   1:  PR[GP1:91,1] = PR[GP1:90,1] + -0.145;
   1:  PR[GP1:91,2] = PR[GP1:90,2] + -15.711;
   1:L PR[91] 10mm/sec CNT100;
   1:  PR[GP1:91,1] = PR[GP1:90,1] + 0.024;
   1:  PR[GP1:91,2] = PR[GP1:90,2] + -15.638;
   1:L PR[91] 10mm/sec CNT100;
   1:  PR[GP1:91,1] = PR[GP1:90,1] + 0.412;
   1:  PR[GP1:91,2] = PR[GP1:90,2] + -15.609;
   1:L PR[91] 10mm/sec CNT100;
   1:  PR[GP1:91,1] = PR[GP1:90,1] + 1.712;
   1:  PR[GP1:91,2] = PR[GP1:90,2] + -16.090;
   1:L PR[91] 10mm/sec CNT100;
   1:  PR[GP1:91,1] = PR[GP1:90,1] + 2.427;
   1:  PR[GP1:91,2] = PR[GP1:90,2] + -16.554;
   1:L PR[91] 10mm/sec CNT100;
   1:  PR[GP1:91,1] = PR[GP1:90,1] + 3.285;
   1:  PR[GP1:91,2] = PR[GP1:90,2] + -17.042;
   1:L PR[91] 10mm/sec CNT100;
   1:  PR[GP1:91,1] = PR[GP1:90,1] + 4.793;
   1:  PR[GP1:91,2] = PR[GP1:90,2] + -17.836;
   1:L PR[91] 10mm/sec CNT100;
   1:  PR[GP1:91,1] = PR[GP1:90,1] + 5.956;
   1:  PR[GP1:91,2] = PR[GP1:90,2] + -18.277;
   1:L PR[91] 10mm/sec CNT100;
   1:  PR[GP1:91,1] = PR[GP1:90,1] + 7.268;
   1:  PR[GP1:91,2] = PR[GP1:90,2] + -18.717;
   1:L PR[91] 10mm/sec CNT100;
   1:  PR[GP1:91,1] = PR[GP1:90,1] + 8.896;
   1:  PR[GP1:91,2] = PR[GP1:90,2] + -19.063;
   1:L PR[91] 10mm/sec CNT100;
   1:  PR[GP1:91,1] = PR[GP1:90,1] + 9.804;
   1:  PR[GP1:91,2] = PR[GP1:90,2] + -19.215;
   1:L PR[91] 10mm/sec CNT100;
   1:  PR[GP1:91,1] = PR[GP1:90,1] + 12.012;
   1:  PR[GP1:91,2] = PR[GP1:90,2] + -19.347;
   1:L PR[91] 10mm/sec CNT100;
   1:  PR[GP1:91,1] = PR[GP1:90,1] + 12.321;
   1:  PR[GP1:91,2] = PR[GP1:90,2] + -19.350;
   1:L PR[91] 10mm/sec CNT100;
   1:  PR[GP1:91,1] = PR[GP1:90,1] + 13.545;
   1:  PR[GP1:91,2] = PR[GP1:90,2] + -19.242;
   1:L PR[91] 10mm/sec CNT100;
   1:  PR[GP1:91,1] = PR[GP1:90,1] + 14.916;
   1:  PR[GP1:91,2] = PR[GP1:90,2] + -19.147;
   1:L PR[91] 10mm/sec CNT100;
   1:  PR[GP1:91,1] = PR[GP1:90,1] + 17.562;
   1:  PR[GP1:91,2] = PR[GP1:90,2] + -18.593;
   1:L PR[91] 10mm/sec CNT100;
   1:  PR[GP1:91,1] = PR[GP1:90,1] + 19.003;
   1:  PR[GP1:91,2] = PR[GP1:90,2] + -18.092;
   1:L PR[91] 10mm/sec CNT100;
   1:  PR[GP1:91,1] = PR[GP1:90,1] + 20.123;
   1:  PR[GP1:91,2] = PR[GP1:90,2] + -17.685;
   1:L PR[91] 10mm/sec CNT100;
   1:  PR[GP1:91,1] = PR[GP1:90,1] + 22.568;
   1:  PR[GP1:91,2] = PR[GP1:90,2] + -16.427;
   1:L PR[91] 10mm/sec CNT100;
   1:  PR[GP1:91,1] = PR[GP1:90,1] + 24.867;
   1:  PR[GP1:91,2] = PR[GP1:90,2] + -14.882;
   1:L PR[91] 10mm/sec CNT100;
   1:  PR[GP1:91,1] = PR[GP1:90,1] + 25.707;
   1:  PR[GP1:91,2] = PR[GP1:90,2] + -14.143;
   1:L PR[91] 10mm/sec CNT100;
   1:  PR[GP1:91,1] = PR[GP1:90,1] + 26.925;
   1:  PR[GP1:91,2] = PR[GP1:90,2] + -13.045;
   1:L PR[91] 10mm/sec CNT100;
   1:  PR[GP1:91,1] = PR[GP1:90,1] + 28.700;
   1:  PR[GP1:91,2] = PR[GP1:90,2] + -10.934;
   1:L PR[91] 10mm/sec CNT100;
   1:  PR[GP1:91,1] = PR[GP1:90,1] + 30.141;
   1:  PR[GP1:91,2] = PR[GP1:90,2] + -8.600;
   1:L PR[91] 10mm/sec CNT100;
   1:  PR[GP1:91,1] = PR[GP1:90,1] + 31.207;
   1:  PR[GP1:91,2] = PR[GP1:90,2] + -6.109;
   1:L PR[91] 10mm/sec CNT100;
   1:  PR[GP1:91,1] = PR[GP1:90,1] + 31.857;
   1:  PR[GP1:91,2] = PR[GP1:90,2] + -3.509;
   1:L PR[91] 10mm/sec CNT100;
   1:  PR[GP1:91,1] = PR[GP1:90,1] + 32.061;
   1:  PR[GP1:91,2] = PR[GP1:90,2] + -0.854;
   1:L PR[91] 10mm/sec CNT100;
   1:  PR[GP1:91,1] = PR[GP1:90,1] + 31.675;
   1:  PR[GP1:91,2] = PR[GP1:90,2] + 2.503;
   1:L PR[91] 10mm/sec CNT100;
   1:  PR[GP1:91,1] = PR[GP1:90,1] + 30.594;
   1:  PR[GP1:91,2] = PR[GP1:90,2] + 5.692;
   1:L PR[91] 10mm/sec CNT100;
   1:  PR[GP1:91,1] = PR[GP1:90,1] + 28.845;
   1:  PR[GP1:91,2] = PR[GP1:90,2] + 8.602;
   1:L PR[91] 10mm/sec CNT100;
   1:  PR[GP1:91,1] = PR[GP1:90,1] + 26.495;
   1:  PR[GP1:91,2] = PR[GP1:90,2] + 11.109;
   1:L PR[91] 10mm/sec CNT100;
   1:  PR[GP1:91,1] = PR[GP1:90,1] + 23.637;
   1:  PR[GP1:91,2] = PR[GP1:90,2] + 13.130;
   1:L PR[91] 10mm/sec CNT100;
   1:  PR[GP1:91,1] = PR[GP1:90,1] + 20.377;
   1:  PR[GP1:91,2] = PR[GP1:90,2] + 14.590;
   1:L PR[91] 10mm/sec CNT100;
   1:  PR[GP1:91,1] = PR[GP1:90,1] + 16.885;
   1:  PR[GP1:91,2] = PR[GP1:90,2] + 15.406;
   1:L PR[91] 10mm/sec CNT100;
   1:  PR[GP1:91,1] = PR[GP1:90,1] + 14.816;
   1:  PR[GP1:91,2] = PR[GP1:90,2] + 15.503;
   1:L PR[91] 10mm/sec CNT100;
   1:  PR[GP1:91,1] = PR[GP1:90,1] + 13.268;
   1:  PR[GP1:91,2] = PR[GP1:90,2] + 15.568;
   1:L PR[91] 10mm/sec CNT100;
   1:  PR[GP1:91,1] = PR[GP1:90,1] + 9.649;
   1:  PR[GP1:91,2] = PR[GP1:90,2] + 15.081;
   1:L PR[91] 10mm/sec CNT100;
   1:  PR[GP1:91,1] = PR[GP1:90,1] + 6.237;
   1:  PR[GP1:91,2] = PR[GP1:90,2] + 13.936;
   1:L PR[91] 10mm/sec CNT100;
   1:  PR[GP1:91,1] = PR[GP1:90,1] + 3.041;
   1:  PR[GP1:91,2] = PR[GP1:90,2] + 12.211;
   1:L PR[91] 10mm/sec CNT100;
   1:  PR[GP1:91,1] = PR[GP1:90,1] + 1.090;
   1:  PR[GP1:91,2] = PR[GP1:90,2] + 10.690;
   1:L PR[91] 10mm/sec CNT100;
   1:  PR[GP1:91,1] = PR[GP1:90,1] + -0.001;
   1:  PR[GP1:91,2] = PR[GP1:90,2] + 10.133;
   1:L PR[91] 10mm/sec CNT100;
   1:  PR[GP1:91,1] = PR[GP1:90,1] + -1.282;
   1:  PR[GP1:91,2] = PR[GP1:90,2] + 10.163;
   1:L PR[91] 10mm/sec CNT100;
   1:  PR[GP1:91,1] = PR[GP1:90,1] + -2.059;
   1:  PR[GP1:91,2] = PR[GP1:90,2] + 10.540;
   1:L PR[91] 10mm/sec CNT100;
   1:  PR[GP1:91,1] = PR[GP1:90,1] + -3.147;
   1:  PR[GP1:91,2] = PR[GP1:90,2] + 11.202;
   1:L PR[91] 10mm/sec CNT100;
   1:  PR[GP1:91,1] = PR[GP1:90,1] + -4.530;
   1:  PR[GP1:91,2] = PR[GP1:90,2] + 12.155;
   1:L PR[91] 10mm/sec CNT100;
   1:  PR[GP1:91,1] = PR[GP1:90,1] + -5.421;
   1:  PR[GP1:91,2] = PR[GP1:90,2] + 12.681;
   1:L PR[91] 10mm/sec CNT100;
   1:  PR[GP1:91,1] = PR[GP1:90,1] + -7.191;
   1:  PR[GP1:91,2] = PR[GP1:90,2] + 13.488;
   1:L PR[91] 10mm/sec CNT100;
   1:  PR[GP1:91,1] = PR[GP1:90,1] + -9.797;
   1:  PR[GP1:91,2] = PR[GP1:90,2] + 14.446;
   1:L PR[91] 10mm/sec CNT100;
   1:  PR[GP1:91,1] = PR[GP1:90,1] + -10.237;
   1:  PR[GP1:91,2] = PR[GP1:90,2] + 14.563;
   1:L PR[91] 10mm/sec CNT100;
   1:  PR[GP1:91,1] = PR[GP1:90,1] + -13.368;
   1:  PR[GP1:91,2] = PR[GP1:90,2] + 15.140;
   1:L PR[91] 10mm/sec CNT100;
   1:  PR[GP1:91,1] = PR[GP1:90,1] + -14.004;
   1:  PR[GP1:91,2] = PR[GP1:90,2] + 15.238;
   1:L PR[91] 10mm/sec CNT100;
   1:  PR[GP1:91,1] = PR[GP1:90,1] + -16.372;
   1:  PR[GP1:91,2] = PR[GP1:90,2] + 15.227;
   1:L PR[91] 10mm/sec CNT100;
   1:  PR[GP1:91,1] = PR[GP1:90,1] + -17.931;
   1:  PR[GP1:91,2] = PR[GP1:90,2] + 15.176;
   1:L PR[91] 10mm/sec CNT100;
   1:  PR[GP1:91,1] = PR[GP1:90,1] + -19.411;
   1:  PR[GP1:91,2] = PR[GP1:90,2] + 14.876;
   1:L PR[91] 10mm/sec CNT100;
   1:  PR[GP1:91,1] = PR[GP1:90,1] + -21.644;
   1:  PR[GP1:91,2] = PR[GP1:90,2] + 14.370;
   1:L PR[91] 10mm/sec CNT100;
   1:  PR[GP1:91,1] = PR[GP1:90,1] + -22.403;
   1:  PR[GP1:91,2] = PR[GP1:90,2] + 14.049;
   1:L PR[91] 10mm/sec CNT100;
   1:  PR[GP1:91,1] = PR[GP1:90,1] + -25.006;
   1:  PR[GP1:91,2] = PR[GP1:90,2] + 12.891;
   1:L PR[91] 10mm/sec CNT100;
   1:  PR[GP1:91,1] = PR[GP1:90,1] + -27.897;
   1:  PR[GP1:91,2] = PR[GP1:90,2] + 10.819;
   1:L PR[91] 10mm/sec CNT100;
   1:  PR[GP1:91,1] = PR[GP1:90,1] + -30.164;
   1:  PR[GP1:91,2] = PR[GP1:90,2] + 8.232;
   1:L PR[91] 10mm/sec CNT100;
   1:  PR[GP1:91,1] = PR[GP1:90,1] + -31.840;
   1:  PR[GP1:91,2] = PR[GP1:90,2] + 5.244;
   1:L PR[91] 10mm/sec CNT100;
   1:  PR[GP1:91,1] = PR[GP1:90,1] + -32.875;
   1:  PR[GP1:91,2] = PR[GP1:90,2] + 1.996;
   1:L PR[91] 10mm/sec CNT100;
   1:  PR[GP1:91,1] = PR[GP1:90,1] + -33.174;
   1:  PR[GP1:91,2] = PR[GP1:90,2] + -1.394;
   1:L PR[91] 10mm/sec CNT100;
   1:  PR[GP1:91,1] = PR[GP1:90,1] + -33.130;
   1:  PR[GP1:91,2] = PR[GP1:90,2] + -1.625;
   1:L PR[91] 10mm/sec CNT100;
   1:  PR[GP1:91,1] = PR[GP1:90,1] + -32.704;
   1:  PR[GP1:91,2] = PR[GP1:90,2] + -4.886;
   1:L PR[91] 10mm/sec CNT100;
   1:  PR[GP1:91,1] = PR[GP1:90,1] + -32.550;
   1:  PR[GP1:91,2] = PR[GP1:90,2] + -5.342;
   1:L PR[91] 10mm/sec CNT100;
   1:  PR[GP1:91,1] = PR[GP1:90,1] + -31.594;
   1:  PR[GP1:91,2] = PR[GP1:90,2] + -7.989;
   1:L PR[91] 10mm/sec CNT100;
   1:  PR[GP1:91,1] = PR[GP1:90,1] + -31.506;
   1:  PR[GP1:91,2] = PR[GP1:90,2] + -8.224;
   1:L PR[91] 10mm/sec CNT100;
   1:  PR[GP1:91,1] = PR[GP1:90,1] + -29.951;
   1:  PR[GP1:91,2] = PR[GP1:90,2] + -10.706;
   1:L PR[91] 10mm/sec CNT100;
   1:  PR[GP1:91,1] = PR[GP1:90,1] + -29.521;
   1:  PR[GP1:91,2] = PR[GP1:90,2] + -11.361;
   1:L PR[91] 10mm/sec CNT100;
   1:  PR[GP1:91,1] = PR[GP1:90,1] + -27.878;
   1:  PR[GP1:91,2] = PR[GP1:90,2] + -13.093;
   1:L PR[91] 10mm/sec CNT100;
   1:  PR[GP1:91,1] = PR[GP1:90,1] + -26.835;
   1:  PR[GP1:91,2] = PR[GP1:90,2] + -14.134;
   1:L PR[91] 10mm/sec CNT100;
   1:  PR[GP1:91,1] = PR[GP1:90,1] + -25.477;
   1:  PR[GP1:91,2] = PR[GP1:90,2] + -15.103;
   1:L PR[91] 10mm/sec CNT100;
   1:  PR[GP1:91,1] = PR[GP1:90,1] + -22.956;
   1:  PR[GP1:91,2] = PR[GP1:90,2] + -16.602;
   1:  PR[GP1:91,3] = PR[GP1:90,3] + 26.400;
   1:L PR[91] 10mm/sec CNT100;
   1:  PR[GP1:91,1] = PR[GP1:90,1] + -19.409;
   1:  PR[GP1:91,2] = PR[GP1:90,2] + -18.084;
   1:L PR[91] 10mm/sec CNT100;
   1:  PR[GP1:91,1] = PR[GP1:90,1] + -17.838;
   1:  PR[GP1:91,2] = PR[GP1:90,2] + -18.496;
   1:L PR[91] 10mm/sec CNT100;
   1:  PR[GP1:91,1] = PR[GP1:90,1] + -15.882;
   1:  PR[GP1:91,2] = PR[GP1:90,2] + -18.925;
   1:L PR[91] 10mm/sec CNT100;
   1:  PR[GP1:91,1] = PR[GP1:90,1] + -12.351;
   1:  PR[GP1:91,2] = PR[GP1:90,2] + -19.223;
   1:L PR[91] 10mm/sec CNT100;
   1:  PR[GP1:91,1] = PR[GP1:90,1] + -9.475;
   1:  PR[GP1:91,2] = PR[GP1:90,2] + -19.059;
   1:L PR[91] 10mm/sec CNT100;
   1:  PR[GP1:91,1] = PR[GP1:90,1] + -8.254;
   1:  PR[GP1:91,2] = PR[GP1:90,2] + -18.972;
   1:L PR[91] 10mm/sec CNT100;
   1:  PR[GP1:91,1] = PR[GP1:90,1] + -5.076;
   1:  PR[GP1:91,2] = PR[GP1:90,2] + -18.282;
   1:L PR[91] 10mm/sec CNT100;
   1:  PR[GP1:91,1] = PR[GP1:90,1] + -2.226;
   1:  PR[GP1:91,2] = PR[GP1:90,2] + -17.323;
   1:L PR[91] 10mm/sec CNT100;
   1:  PR[GP1:91,1] = PR[GP1:90,1] + -1.447;
   1:  PR[GP1:91,2] = PR[GP1:90,2] + -16.960;
   1:L PR[91] 10mm/sec CNT100;
   1:  PR[GP1:91,1] = PR[GP1:90,1] + -0.532;
   1:  PR[GP1:91,2] = PR[GP1:90,2] + -16.498;
   1:L PR[91] 10mm/sec CNT100;
   1:  PR[GP1:91,1] = PR[GP1:90,1] + 0.549;
   1:  PR[GP1:91,2] = PR[GP1:90,2] + -16.236;
   1:L PR[91] 10mm/sec CNT100;
   1:  PR[GP1:91,1] = PR[GP1:90,1] + 1.911;
   1:  PR[GP1:91,2] = PR[GP1:90,2] + -16.677;
   1:L PR[91] 10mm/sec CNT100;
   1:  PR[GP1:91,1] = PR[GP1:90,1] + 2.459;
   1:  PR[GP1:91,2] = PR[GP1:90,2] + -17.007;
   1:L PR[91] 10mm/sec CNT100;
   1:  PR[GP1:91,1] = PR[GP1:90,1] + 4.600;
   1:  PR[GP1:91,2] = PR[GP1:90,2] + -18.134;
   1:L PR[91] 10mm/sec CNT100;
   1:  PR[GP1:91,1] = PR[GP1:90,1] + 5.082;
   1:  PR[GP1:91,2] = PR[GP1:90,2] + -18.317;
   1:L PR[91] 10mm/sec CNT100;
   1:  PR[GP1:91,1] = PR[GP1:90,1] + 7.132;
   1:  PR[GP1:91,2] = PR[GP1:90,2] + -19.005;
   1:L PR[91] 10mm/sec CNT100;
   1:  PR[GP1:91,1] = PR[GP1:90,1] + 7.995;
   1:  PR[GP1:91,2] = PR[GP1:90,2] + -19.188;
   1:L PR[91] 10mm/sec CNT100;
   1:  PR[GP1:91,1] = PR[GP1:90,1] + 9.727;
   1:  PR[GP1:91,2] = PR[GP1:90,2] + -19.478;
   1:L PR[91] 10mm/sec CNT100;
   1:  PR[GP1:91,1] = PR[GP1:90,1] + 11.103;
   1:  PR[GP1:91,2] = PR[GP1:90,2] + -19.560;
   1:L PR[91] 10mm/sec CNT100;
   1:  PR[GP1:91,1] = PR[GP1:90,1] + 12.304;
   1:  PR[GP1:91,2] = PR[GP1:90,2] + -19.572;
   1:L PR[91] 10mm/sec CNT100;
   1:  PR[GP1:91,1] = PR[GP1:90,1] + 14.298;
   1:  PR[GP1:91,2] = PR[GP1:90,2] + -19.396;
   1:L PR[91] 10mm/sec CNT100;
   1:  PR[GP1:91,1] = PR[GP1:90,1] + 14.791;
   1:  PR[GP1:91,2] = PR[GP1:90,2] + -19.325;
   1:L PR[91] 10mm/sec CNT100;
   1:  PR[GP1:91,1] = PR[GP1:90,1] + 16.410;
   1:  PR[GP1:91,2] = PR[GP1:90,2] + -18.940;
   1:L PR[91] 10mm/sec CNT100;
   1:  PR[GP1:91,1] = PR[GP1:90,1] + 17.275;
   1:  PR[GP1:91,2] = PR[GP1:90,2] + -18.756;
   1:L PR[91] 10mm/sec CNT100;
   1:  PR[GP1:91,1] = PR[GP1:90,1] + 19.829;
   1:  PR[GP1:91,2] = PR[GP1:90,2] + -17.832;
   1:L PR[91] 10mm/sec CNT100;
   1:  PR[GP1:91,1] = PR[GP1:90,1] + 22.250;
   1:  PR[GP1:91,2] = PR[GP1:90,2] + -16.569;
   1:L PR[91] 10mm/sec CNT100;
   1:  PR[GP1:91,1] = PR[GP1:90,1] + 24.493;
   1:  PR[GP1:91,2] = PR[GP1:90,2] + -14.979;
   1:L PR[91] 10mm/sec CNT100;
   1:  PR[GP1:91,1] = PR[GP1:90,1] + 26.536;
   1:  PR[GP1:91,2] = PR[GP1:90,2] + -13.129;
   1:L PR[91] 10mm/sec CNT100;
   1:  PR[GP1:91,1] = PR[GP1:90,1] + 28.291;
   1:  PR[GP1:91,2] = PR[GP1:90,2] + -11.021;
   1:L PR[91] 10mm/sec CNT100;
   1:  PR[GP1:91,1] = PR[GP1:90,1] + 29.712;
   1:  PR[GP1:91,2] = PR[GP1:90,2] + -8.689;
   1:L PR[91] 10mm/sec CNT100;
   1:  PR[GP1:91,1] = PR[GP1:90,1] + 30.692;
   1:  PR[GP1:91,2] = PR[GP1:90,2] + -6.354;
   1:L PR[91] 10mm/sec CNT100;
   1:  PR[GP1:91,1] = PR[GP1:90,1] + 30.760;
   1:  PR[GP1:91,2] = PR[GP1:90,2] + -6.189;
   1:L PR[91] 10mm/sec CNT100;
   1:  PR[GP1:91,1] = PR[GP1:90,1] + 31.399;
   1:  PR[GP1:91,2] = PR[GP1:90,2] + -3.584;
   1:L PR[91] 10mm/sec CNT100;
   1:  PR[GP1:91,1] = PR[GP1:90,1] + 31.597;
   1:  PR[GP1:91,2] = PR[GP1:90,2] + -0.937;
   1:L PR[91] 10mm/sec CNT100;
   1:  PR[GP1:91,1] = PR[GP1:90,1] + 31.211;
   1:  PR[GP1:91,2] = PR[GP1:90,2] + 2.414;
   1:L PR[91] 10mm/sec CNT100;
   1:  PR[GP1:91,1] = PR[GP1:90,1] + 30.126;
   1:  PR[GP1:91,2] = PR[GP1:90,2] + 5.602;
   1:L PR[91] 10mm/sec CNT100;
   1:  PR[GP1:91,1] = PR[GP1:90,1] + 28.371;
   1:  PR[GP1:91,2] = PR[GP1:90,2] + 8.503;
   1:L PR[91] 10mm/sec CNT100;
   1:  PR[GP1:91,1] = PR[GP1:90,1] + 26.016;
   1:  PR[GP1:91,2] = PR[GP1:90,2] + 11.013;
   1:L PR[91] 10mm/sec CNT100;
   1:  PR[GP1:91,1] = PR[GP1:90,1] + 23.154;
   1:  PR[GP1:91,2] = PR[GP1:90,2] + 13.036;
   1:L PR[91] 10mm/sec CNT100;
   1:  PR[GP1:91,1] = PR[GP1:90,1] + 19.918;
   1:  PR[GP1:91,2] = PR[GP1:90,2] + 14.479;
   1:L PR[91] 10mm/sec CNT100;
   1:  PR[GP1:91,1] = PR[GP1:90,1] + 16.430;
   1:  PR[GP1:91,2] = PR[GP1:90,2] + 15.290;
   1:L PR[91] 10mm/sec CNT100;
   1:  PR[GP1:91,1] = PR[GP1:90,1] + 15.306;
   1:  PR[GP1:91,2] = PR[GP1:90,2] + 15.342;
   1:L PR[91] 10mm/sec CNT100;
   1:  PR[GP1:91,1] = PR[GP1:90,1] + 12.826;
   1:  PR[GP1:91,2] = PR[GP1:90,2] + 15.446;
   1:L PR[91] 10mm/sec CNT100;
   1:  PR[GP1:91,1] = PR[GP1:90,1] + 11.054;
   1:  PR[GP1:91,2] = PR[GP1:90,2] + 15.211;
   1:L PR[91] 10mm/sec CNT100;
   1:  PR[GP1:91,1] = PR[GP1:90,1] + 9.258;
   1:  PR[GP1:91,2] = PR[GP1:90,2] + 14.945;
   1:L PR[91] 10mm/sec CNT100;
   1:  PR[GP1:91,1] = PR[GP1:90,1] + 5.841;
   1:  PR[GP1:91,2] = PR[GP1:90,2] + 13.802;
   1:L PR[91] 10mm/sec CNT100;
   1:  PR[GP1:91,1] = PR[GP1:90,1] + 3.815;
   1:  PR[GP1:91,2] = PR[GP1:90,2] + 12.709;
   1:L PR[91] 10mm/sec CNT100;
   1:  PR[GP1:91,1] = PR[GP1:90,1] + 2.698;
   1:  PR[GP1:91,2] = PR[GP1:90,2] + 12.073;
   1:L PR[91] 10mm/sec CNT100;
   1:  PR[GP1:91,1] = PR[GP1:90,1] + 1.151;
   1:  PR[GP1:91,2] = PR[GP1:90,2] + 10.923;
   1:L PR[91] 10mm/sec CNT100;
   1:  PR[GP1:91,1] = PR[GP1:90,1] + 0.972;
   1:  PR[GP1:91,2] = PR[GP1:90,2] + 10.850;
   1:L PR[91] 10mm/sec CNT100;
   1:  PR[GP1:91,1] = PR[GP1:90,1] + 0.160;
   1:  PR[GP1:91,2] = PR[GP1:90,2] + 10.403;
   1:L PR[91] 10mm/sec CNT100;
   1:  PR[GP1:91,1] = PR[GP1:90,1] + -0.093;
   1:  PR[GP1:91,2] = PR[GP1:90,2] + 10.374;
   1:L PR[91] 10mm/sec CNT100;
   1:  PR[GP1:91,1] = PR[GP1:90,1] + -0.386;
   1:  PR[GP1:91,2] = PR[GP1:90,2] + 10.415;
   1:L PR[91] 10mm/sec CNT100;
   1:  PR[GP1:91,1] = PR[GP1:90,1] + -1.188;
   1:  PR[GP1:91,2] = PR[GP1:90,2] + 10.429;
   1:L PR[91] 10mm/sec CNT100;
   1:  PR[GP1:91,1] = PR[GP1:90,1] + -1.894;
   1:  PR[GP1:91,2] = PR[GP1:90,2] + 10.798;
   1:L PR[91] 10mm/sec CNT100;
   1:  PR[GP1:91,1] = PR[GP1:90,1] + -4.413;
   1:  PR[GP1:91,2] = PR[GP1:90,2] + 12.333;
   1:L PR[91] 10mm/sec CNT100;
   1:  PR[GP1:91,1] = PR[GP1:90,1] + -7.064;
   1:  PR[GP1:91,2] = PR[GP1:90,2] + 13.542;
   1:L PR[91] 10mm/sec CNT100;
   1:  PR[GP1:91,1] = PR[GP1:90,1] + -8.711;
   1:  PR[GP1:91,2] = PR[GP1:90,2] + 14.147;
   1:L PR[91] 10mm/sec CNT100;
   1:  PR[GP1:91,1] = PR[GP1:90,1] + -10.068;
   1:  PR[GP1:91,2] = PR[GP1:90,2] + 14.509;
   1:L PR[91] 10mm/sec CNT100;
   1:  PR[GP1:91,1] = PR[GP1:90,1] + -13.422;
   1:  PR[GP1:91,2] = PR[GP1:90,2] + 15.102;
   1:L PR[91] 10mm/sec CNT100;
   1:  PR[GP1:91,1] = PR[GP1:90,1] + -16.470;
   1:  PR[GP1:91,2] = PR[GP1:90,2] + 15.087;
   1:L PR[91] 10mm/sec CNT100;
   1:  PR[GP1:91,1] = PR[GP1:90,1] + -17.366;
   1:  PR[GP1:91,2] = PR[GP1:90,2] + 15.058;
   1:L PR[91] 10mm/sec CNT100;
   1:  PR[GP1:91,1] = PR[GP1:90,1] + -19.480;
   1:  PR[GP1:91,2] = PR[GP1:90,2] + 14.630;
   1:L PR[91] 10mm/sec CNT100;
   1:  PR[GP1:91,1] = PR[GP1:90,1] + -21.106;
   1:  PR[GP1:91,2] = PR[GP1:90,2] + 14.262;
   1:L PR[91] 10mm/sec CNT100;
   1:  PR[GP1:91,1] = PR[GP1:90,1] + -22.430;
   1:  PR[GP1:91,2] = PR[GP1:90,2] + 13.703;
   1:L PR[91] 10mm/sec CNT100;
   1:  PR[GP1:91,1] = PR[GP1:90,1] + -24.497;
   1:  PR[GP1:91,2] = PR[GP1:90,2] + 12.783;
   1:L PR[91] 10mm/sec CNT100;
   1:  PR[GP1:91,1] = PR[GP1:90,1] + -25.221;
   1:  PR[GP1:91,2] = PR[GP1:90,2] + 12.281;
   1:L PR[91] 10mm/sec CNT100;
   1:  PR[GP1:91,1] = PR[GP1:90,1] + -27.417;
   1:  PR[GP1:91,2] = PR[GP1:90,2] + 10.708;
   1:L PR[91] 10mm/sec CNT100;
   1:  PR[GP1:91,1] = PR[GP1:90,1] + -29.766;
   1:  PR[GP1:91,2] = PR[GP1:90,2] + 8.122;
   1:L PR[91] 10mm/sec CNT100;
   1:  PR[GP1:91,1] = PR[GP1:90,1] + -31.480;
   1:  PR[GP1:91,2] = PR[GP1:90,2] + 5.138;
   1:L PR[91] 10mm/sec CNT100;
   1:  PR[GP1:91,1] = PR[GP1:90,1] + -32.520;
   1:  PR[GP1:91,2] = PR[GP1:90,2] + 1.891;
   1:L PR[91] 10mm/sec CNT100;
   1:  PR[GP1:91,1] = PR[GP1:90,1] + -32.766;
   1:  PR[GP1:91,2] = PR[GP1:90,2] + -1.539;
   1:L PR[91] 10mm/sec CNT100;
   1:  PR[GP1:91,1] = PR[GP1:90,1] + -32.245;
   1:  PR[GP1:91,2] = PR[GP1:90,2] + -5.041;
   1:L PR[91] 10mm/sec CNT100;
   1:  PR[GP1:91,1] = PR[GP1:90,1] + -31.014;
   1:  PR[GP1:91,2] = PR[GP1:90,2] + -8.415;
   1:L PR[91] 10mm/sec CNT100;
   1:  PR[GP1:91,1] = PR[GP1:90,1] + -29.773;
   1:  PR[GP1:91,2] = PR[GP1:90,2] + -10.397;
   1:L PR[91] 10mm/sec CNT100;
   1:  PR[GP1:91,1] = PR[GP1:90,1] + -29.006;
   1:  PR[GP1:91,2] = PR[GP1:90,2] + -11.565;
   1:L PR[91] 10mm/sec CNT100;
   1:  PR[GP1:91,1] = PR[GP1:90,1] + -27.788;
   1:  PR[GP1:91,2] = PR[GP1:90,2] + -12.849;
   1:L PR[91] 10mm/sec CNT100;
   1:  PR[GP1:91,1] = PR[GP1:90,1] + -26.287;
   1:  PR[GP1:91,2] = PR[GP1:90,2] + -14.347;
   1:L PR[91] 10mm/sec CNT100;
   1:  PR[GP1:91,1] = PR[GP1:90,1] + -25.464;
   1:  PR[GP1:91,2] = PR[GP1:90,2] + -14.935;
   1:L PR[91] 10mm/sec CNT100;
   1:  PR[GP1:91,1] = PR[GP1:90,1] + -24.303;
   1:  PR[GP1:91,2] = PR[GP1:90,2] + -15.530;
   1:  PR[GP1:91,3] = PR[GP1:90,3] + 27.500;
   1:L PR[91] 10mm/sec CNT100;
   1:  PR[GP1:91,1] = PR[GP1:90,1] + -22.470;
   1:  PR[GP1:91,2] = PR[GP1:90,2] + -16.723;
   1:L PR[91] 10mm/sec CNT100;
   1:  PR[GP1:91,1] = PR[GP1:90,1] + -21.655;
   1:  PR[GP1:91,2] = PR[GP1:90,2] + -17.097;
   1:L PR[91] 10mm/sec CNT100;
   1:  PR[GP1:91,1] = PR[GP1:90,1] + -19.019;
   1:  PR[GP1:91,2] = PR[GP1:90,2] + -18.195;
   1:L PR[91] 10mm/sec CNT100;
   1:  PR[GP1:91,1] = PR[GP1:90,1] + -16.269;
   1:  PR[GP1:91,2] = PR[GP1:90,2] + -18.917;
   1:L PR[91] 10mm/sec CNT100;
   1:  PR[GP1:91,1] = PR[GP1:90,1] + -15.563;
   1:  PR[GP1:91,2] = PR[GP1:90,2] + -19.071;
   1:L PR[91] 10mm/sec CNT100;
   1:  PR[GP1:91,1] = PR[GP1:90,1] + -14.385;
   1:  PR[GP1:91,2] = PR[GP1:90,2] + -19.169;
   1:L PR[91] 10mm/sec CNT100;
   1:  PR[GP1:91,1] = PR[GP1:90,1] + -12.195;
   1:  PR[GP1:91,2] = PR[GP1:90,2] + -19.412;
   1:L PR[91] 10mm/sec CNT100;
   1:  PR[GP1:91,1] = PR[GP1:90,1] + -11.314;
   1:  PR[GP1:91,2] = PR[GP1:90,2] + -19.461;
   1:L PR[91] 10mm/sec CNT100;
   1:  PR[GP1:91,1] = PR[GP1:90,1] + -9.397;
   1:  PR[GP1:91,2] = PR[GP1:90,2] + -19.352;
   1:L PR[91] 10mm/sec CNT100;
   1:  PR[GP1:91,1] = PR[GP1:90,1] + -7.471;
   1:  PR[GP1:91,2] = PR[GP1:90,2] + -19.215;
   1:L PR[91] 10mm/sec CNT100;
   1:  PR[GP1:91,1] = PR[GP1:90,1] + -6.428;
   1:  PR[GP1:91,2] = PR[GP1:90,2] + -18.988;
   1:L PR[91] 10mm/sec CNT100;
   1:  PR[GP1:91,1] = PR[GP1:90,1] + -4.152;
   1:  PR[GP1:91,2] = PR[GP1:90,2] + -18.587;
   1:L PR[91] 10mm/sec CNT100;
   1:  PR[GP1:91,1] = PR[GP1:90,1] + -1.604;
   1:  PR[GP1:91,2] = PR[GP1:90,2] + -17.734;
   1:L PR[91] 10mm/sec CNT100;
   1:  PR[GP1:91,1] = PR[GP1:90,1] + -0.960;
   1:  PR[GP1:91,2] = PR[GP1:90,2] + -17.455;
   1:L PR[91] 10mm/sec CNT100;
   1:  PR[GP1:91,1] = PR[GP1:90,1] + -0.198;
   1:  PR[GP1:91,2] = PR[GP1:90,2] + -17.088;
   1:L PR[91] 10mm/sec CNT100;
   1:  PR[GP1:91,1] = PR[GP1:90,1] + 0.752;
   1:  PR[GP1:91,2] = PR[GP1:90,2] + -16.862;
   1:L PR[91] 10mm/sec CNT100;
   1:  PR[GP1:91,1] = PR[GP1:90,1] + 2.107;
   1:  PR[GP1:91,2] = PR[GP1:90,2] + -17.241;
   1:L PR[91] 10mm/sec CNT100;
   1:  PR[GP1:91,1] = PR[GP1:90,1] + 4.377;
   1:  PR[GP1:91,2] = PR[GP1:90,2] + -18.414;
   1:L PR[91] 10mm/sec CNT100;
   1:  PR[GP1:91,1] = PR[GP1:90,1] + 6.995;
   1:  PR[GP1:91,2] = PR[GP1:90,2] + -19.292;
   1:L PR[91] 10mm/sec CNT100;
   1:  PR[GP1:91,1] = PR[GP1:90,1] + 7.094;
   1:  PR[GP1:91,2] = PR[GP1:90,2] + -19.313;
   1:L PR[91] 10mm/sec CNT100;
   1:  PR[GP1:91,1] = PR[GP1:90,1] + 9.650;
   1:  PR[GP1:91,2] = PR[GP1:90,2] + -19.740;
   1:L PR[91] 10mm/sec CNT100;
   1:  PR[GP1:91,1] = PR[GP1:90,1] + 10.195;
   1:  PR[GP1:91,2] = PR[GP1:90,2] + -19.773;
   1:L PR[91] 10mm/sec CNT100;
   1:  PR[GP1:91,1] = PR[GP1:90,1] + 12.286;
   1:  PR[GP1:91,2] = PR[GP1:90,2] + -19.794;
   1:L PR[91] 10mm/sec CNT100;
   1:  PR[GP1:91,1] = PR[GP1:90,1] + 13.404;
   1:  PR[GP1:91,2] = PR[GP1:90,2] + -19.695;
   1:L PR[91] 10mm/sec CNT100;
   1:  PR[GP1:91,1] = PR[GP1:90,1] + 14.829;
   1:  PR[GP1:91,2] = PR[GP1:90,2] + -19.490;
   1:L PR[91] 10mm/sec CNT100;
   1:  PR[GP1:91,1] = PR[GP1:90,1] + 16.592;
   1:  PR[GP1:91,2] = PR[GP1:90,2] + -19.070;
   1:L PR[91] 10mm/sec CNT100;
   1:  PR[GP1:91,1] = PR[GP1:90,1] + 17.219;
   1:  PR[GP1:91,2] = PR[GP1:90,2] + -18.880;
   1:L PR[91] 10mm/sec CNT100;
   1:  PR[GP1:91,1] = PR[GP1:90,1] + 19.044;
   1:  PR[GP1:91,2] = PR[GP1:90,2] + -18.158;
   1:L PR[91] 10mm/sec CNT100;
   1:  PR[GP1:91,1] = PR[GP1:90,1] + 19.533;
   1:  PR[GP1:91,2] = PR[GP1:90,2] + -17.980;
   1:L PR[91] 10mm/sec CNT100;
   1:  PR[GP1:91,1] = PR[GP1:90,1] + 21.939;
   1:  PR[GP1:91,2] = PR[GP1:90,2] + -16.707;
   1:L PR[91] 10mm/sec CNT100;
   1:  PR[GP1:91,1] = PR[GP1:90,1] + 24.161;
   1:  PR[GP1:91,2] = PR[GP1:90,2] + -15.115;
   1:L PR[91] 10mm/sec CNT100;
   1:  PR[GP1:91,1] = PR[GP1:90,1] + 26.145;
   1:  PR[GP1:91,2] = PR[GP1:90,2] + -13.231;
   1:L PR[91] 10mm/sec CNT100;
   1:  PR[GP1:91,1] = PR[GP1:90,1] + 26.470;
   1:  PR[GP1:91,2] = PR[GP1:90,2] + -12.817;
   1:L PR[91] 10mm/sec CNT100;
   1:  PR[GP1:91,1] = PR[GP1:90,1] + 27.882;
   1:  PR[GP1:91,2] = PR[GP1:90,2] + -11.107;
   1:L PR[91] 10mm/sec CNT100;
   1:  PR[GP1:91,1] = PR[GP1:90,1] + 29.288;
   1:  PR[GP1:91,2] = PR[GP1:90,2] + -8.782;
   1:L PR[91] 10mm/sec CNT100;
   1:  PR[GP1:91,1] = PR[GP1:90,1] + 29.847;
   1:  PR[GP1:91,2] = PR[GP1:90,2] + -7.448;
   1:L PR[91] 10mm/sec CNT100;
   1:  PR[GP1:91,1] = PR[GP1:90,1] + 30.322;
   1:  PR[GP1:91,2] = PR[GP1:90,2] + -6.292;
   1:L PR[91] 10mm/sec CNT100;
   1:  PR[GP1:91,1] = PR[GP1:90,1] + 30.951;
   1:  PR[GP1:91,2] = PR[GP1:90,2] + -3.693;
   1:L PR[91] 10mm/sec CNT100;
   1:  PR[GP1:91,1] = PR[GP1:90,1] + 31.132;
   1:  PR[GP1:91,2] = PR[GP1:90,2] + -1.047;
   1:L PR[91] 10mm/sec CNT100;
   1:  PR[GP1:91,1] = PR[GP1:90,1] + 30.744;
   1:  PR[GP1:91,2] = PR[GP1:90,2] + 2.310;
   1:L PR[91] 10mm/sec CNT100;
   1:  PR[GP1:91,1] = PR[GP1:90,1] + 29.656;
   1:  PR[GP1:91,2] = PR[GP1:90,2] + 5.500;
   1:L PR[91] 10mm/sec CNT100;
   1:  PR[GP1:91,1] = PR[GP1:90,1] + 27.897;
   1:  PR[GP1:91,2] = PR[GP1:90,2] + 8.405;
   1:L PR[91] 10mm/sec CNT100;
   1:  PR[GP1:91,1] = PR[GP1:90,1] + 25.537;
   1:  PR[GP1:91,2] = PR[GP1:90,2] + 10.918;
   1:L PR[91] 10mm/sec CNT100;
   1:  PR[GP1:91,1] = PR[GP1:90,1] + 22.688;
   1:  PR[GP1:91,2] = PR[GP1:90,2] + 12.929;
   1:L PR[91] 10mm/sec CNT100;
   1:  PR[GP1:91,1] = PR[GP1:90,1] + 19.475;
   1:  PR[GP1:91,2] = PR[GP1:90,2] + 14.355;
   1:L PR[91] 10mm/sec CNT100;
   1:  PR[GP1:91,1] = PR[GP1:90,1] + 15.974;
   1:  PR[GP1:91,2] = PR[GP1:90,2] + 15.173;
   1:L PR[91] 10mm/sec CNT100;
   1:  PR[GP1:91,1] = PR[GP1:90,1] + 15.797;
   1:  PR[GP1:91,2] = PR[GP1:90,2] + 15.182;
   1:L PR[91] 10mm/sec CNT100;
   1:  PR[GP1:91,1] = PR[GP1:90,1] + 12.389;
   1:  PR[GP1:91,2] = PR[GP1:90,2] + 15.325;
   1:L PR[91] 10mm/sec CNT100;
   1:  PR[GP1:91,1] = PR[GP1:90,1] + 8.862;
   1:  PR[GP1:91,2] = PR[GP1:90,2] + 14.808;
   1:L PR[91] 10mm/sec CNT100;
   1:  PR[GP1:91,1] = PR[GP1:90,1] + 5.444;
   1:  PR[GP1:91,2] = PR[GP1:90,2] + 13.668;
   1:L PR[91] 10mm/sec CNT100;
   1:  PR[GP1:91,1] = PR[GP1:90,1] + 4.591;
   1:  PR[GP1:91,2] = PR[GP1:90,2] + 13.207;
   1:L PR[91] 10mm/sec CNT100;
   1:  PR[GP1:91,1] = PR[GP1:90,1] + 2.334;
   1:  PR[GP1:91,2] = PR[GP1:90,2] + 11.920;
   1:L PR[91] 10mm/sec CNT100;
   1:  PR[GP1:91,1] = PR[GP1:90,1] + 2.181;
   1:  PR[GP1:91,2] = PR[GP1:90,2] + 11.825;
   1:L PR[91] 10mm/sec CNT100;
   1:  PR[GP1:91,1] = PR[GP1:90,1] + 1.268;
   1:  PR[GP1:91,2] = PR[GP1:90,2] + 11.139;
   1:L PR[91] 10mm/sec CNT100;
   1:  PR[GP1:91,1] = PR[GP1:90,1] + 0.807;
   1:  PR[GP1:91,2] = PR[GP1:90,2] + 10.950;
   1:L PR[91] 10mm/sec CNT100;
   1:  PR[GP1:91,1] = PR[GP1:90,1] + 0.260;
   1:  PR[GP1:91,2] = PR[GP1:90,2] + 10.649;
   1:L PR[91] 10mm/sec CNT100;
   1:  PR[GP1:91,1] = PR[GP1:90,1] + -0.026;
   1:  PR[GP1:91,2] = PR[GP1:90,2] + 10.616;
   1:L PR[91] 10mm/sec CNT100;
   1:  PR[GP1:91,1] = PR[GP1:90,1] + -0.522;
   1:  PR[GP1:91,2] = PR[GP1:90,2] + 10.686;
   1:L PR[91] 10mm/sec CNT100;
   1:  PR[GP1:91,1] = PR[GP1:90,1] + -1.087;
   1:  PR[GP1:91,2] = PR[GP1:90,2] + 10.696;
   1:L PR[91] 10mm/sec CNT100;
   1:  PR[GP1:91,1] = PR[GP1:90,1] + -1.696;
   1:  PR[GP1:91,2] = PR[GP1:90,2] + 11.017;
   1:L PR[91] 10mm/sec CNT100;
   1:  PR[GP1:91,1] = PR[GP1:90,1] + -3.338;
   1:  PR[GP1:91,2] = PR[GP1:90,2] + 12.009;
   1:L PR[91] 10mm/sec CNT100;
   1:  PR[GP1:91,1] = PR[GP1:90,1] + -3.998;
   1:  PR[GP1:91,2] = PR[GP1:90,2] + 12.333;
   1:L PR[91] 10mm/sec CNT100;
   1:  PR[GP1:91,1] = PR[GP1:90,1] + -5.724;
   1:  PR[GP1:91,2] = PR[GP1:90,2] + 13.043;
   1:L PR[91] 10mm/sec CNT100;
   1:  PR[GP1:91,1] = PR[GP1:90,1] + -6.937;
   1:  PR[GP1:91,2] = PR[GP1:90,2] + 13.595;
   1:L PR[91] 10mm/sec CNT100;
   1:  PR[GP1:91,1] = PR[GP1:90,1] + -7.624;
   1:  PR[GP1:91,2] = PR[GP1:90,2] + 13.848;
   1:L PR[91] 10mm/sec CNT100;
   1:  PR[GP1:91,1] = PR[GP1:90,1] + -9.902;
   1:  PR[GP1:91,2] = PR[GP1:90,2] + 14.456;
   1:L PR[91] 10mm/sec CNT100;
   1:  PR[GP1:91,1] = PR[GP1:90,1] + -12.305;
   1:  PR[GP1:91,2] = PR[GP1:90,2] + 14.881;
   1:L PR[91] 10mm/sec CNT100;
   1:  PR[GP1:91,1] = PR[GP1:90,1] + -13.173;
   1:  PR[GP1:91,2] = PR[GP1:90,2] + 14.961;
   1:L PR[91] 10mm/sec CNT100;
   1:  PR[GP1:91,1] = PR[GP1:90,1] + -16.810;
   1:  PR[GP1:91,2] = PR[GP1:90,2] + 14.939;
   1:L PR[91] 10mm/sec CNT100;
   1:  PR[GP1:91,1] = PR[GP1:90,1] + -19.550;
   1:  PR[GP1:91,2] = PR[GP1:90,2] + 14.385;
   1:L PR[91] 10mm/sec CNT100;
   1:  PR[GP1:91,1] = PR[GP1:90,1] + -20.568;
   1:  PR[GP1:91,2] = PR[GP1:90,2] + 14.154;
   1:L PR[91] 10mm/sec CNT100;
   1:  PR[GP1:91,1] = PR[GP1:90,1] + -22.457;
   1:  PR[GP1:91,2] = PR[GP1:90,2] + 13.356;
   1:L PR[91] 10mm/sec CNT100;
   1:  PR[GP1:91,1] = PR[GP1:90,1] + -23.982;
   1:  PR[GP1:91,2] = PR[GP1:90,2] + 12.678;
   1:L PR[91] 10mm/sec CNT100;
   1:  PR[GP1:91,1] = PR[GP1:90,1] + -25.192;
   1:  PR[GP1:91,2] = PR[GP1:90,2] + 11.838;
   1:L PR[91] 10mm/sec CNT100;
   1:  PR[GP1:91,1] = PR[GP1:90,1] + -26.922;
   1:  PR[GP1:91,2] = PR[GP1:90,2] + 10.598;
   1:L PR[91] 10mm/sec CNT100;
   1:  PR[GP1:91,1] = PR[GP1:90,1] + -29.286;
   1:  PR[GP1:91,2] = PR[GP1:90,2] + 8.005;
   1:L PR[91] 10mm/sec CNT100;
   1:  PR[GP1:91,1] = PR[GP1:90,1] + -31.009;
   1:  PR[GP1:91,2] = PR[GP1:90,2] + 5.010;
   1:L PR[91] 10mm/sec CNT100;
   1:  PR[GP1:91,1] = PR[GP1:90,1] + -32.056;
   1:  PR[GP1:91,2] = PR[GP1:90,2] + 1.752;
   1:L PR[91] 10mm/sec CNT100;
   1:  PR[GP1:91,1] = PR[GP1:90,1] + -32.299;
   1:  PR[GP1:91,2] = PR[GP1:90,2] + -1.694;
   1:L PR[91] 10mm/sec CNT100;
   1:  PR[GP1:91,1] = PR[GP1:90,1] + -31.934;
   1:  PR[GP1:91,2] = PR[GP1:90,2] + -4.177;
   1:L PR[91] 10mm/sec CNT100;
   1:  PR[GP1:91,1] = PR[GP1:90,1] + -31.769;
   1:  PR[GP1:91,2] = PR[GP1:90,2] + -5.212;
   1:L PR[91] 10mm/sec CNT100;
   1:  PR[GP1:91,1] = PR[GP1:90,1] + -31.026;
   1:  PR[GP1:91,2] = PR[GP1:90,2] + -7.270;
   1:L PR[91] 10mm/sec CNT100;
   1:  PR[GP1:91,1] = PR[GP1:90,1] + -30.526;
   1:  PR[GP1:91,2] = PR[GP1:90,2] + -8.602;
   1:L PR[91] 10mm/sec CNT100;
   1:  PR[GP1:91,1] = PR[GP1:90,1] + -29.595;
   1:  PR[GP1:91,2] = PR[GP1:90,2] + -10.089;
   1:L PR[91] 10mm/sec CNT100;
   1:  PR[GP1:91,1] = PR[GP1:90,1] + -28.492;
   1:  PR[GP1:91,2] = PR[GP1:90,2] + -11.768;
   1:L PR[91] 10mm/sec CNT100;
   1:  PR[GP1:91,1] = PR[GP1:90,1] + -27.698;
   1:  PR[GP1:91,2] = PR[GP1:90,2] + -12.605;
   1:L PR[91] 10mm/sec CNT100;
   1:  PR[GP1:91,1] = PR[GP1:90,1] + -25.739;
   1:  PR[GP1:91,2] = PR[GP1:90,2] + -14.560;
   1:L PR[91] 10mm/sec CNT100;
   1:  PR[GP1:91,1] = PR[GP1:90,1] + -25.450;
   1:  PR[GP1:91,2] = PR[GP1:90,2] + -14.767;
   1:L PR[91] 10mm/sec CNT100;
   1:  PR[GP1:91,1] = PR[GP1:90,1] + -24.946;
   1:  PR[GP1:91,2] = PR[GP1:90,2] + -14.909;
   1:  PR[GP1:91,3] = PR[GP1:90,3] + 28.600;
   1:L PR[91] 10mm/sec CNT100;
   1:  PR[GP1:91,1] = PR[GP1:90,1] + -22.013;
   1:  PR[GP1:91,2] = PR[GP1:90,2] + -16.820;
   1:L PR[91] 10mm/sec CNT100;
   1:  PR[GP1:91,1] = PR[GP1:90,1] + -20.151;
   1:  PR[GP1:91,2] = PR[GP1:90,2] + -17.672;
   1:L PR[91] 10mm/sec CNT100;
   1:  PR[GP1:91,1] = PR[GP1:90,1] + -18.628;
   1:  PR[GP1:91,2] = PR[GP1:90,2] + -18.307;
   1:L PR[91] 10mm/sec CNT100;
   1:  PR[GP1:91,1] = PR[GP1:90,1] + -15.161;
   1:  PR[GP1:91,2] = PR[GP1:90,2] + -19.227;
   1:L PR[91] 10mm/sec CNT100;
   1:  PR[GP1:91,1] = PR[GP1:90,1] + -14.848;
   1:  PR[GP1:91,2] = PR[GP1:90,2] + -19.284;
   1:L PR[91] 10mm/sec CNT100;
   1:  PR[GP1:91,1] = PR[GP1:90,1] + -11.959;
   1:  PR[GP1:91,2] = PR[GP1:90,2] + -19.605;
   1:L PR[91] 10mm/sec CNT100;
   1:  PR[GP1:91,1] = PR[GP1:90,1] + -10.269;
   1:  PR[GP1:91,2] = PR[GP1:90,2] + -19.698;
   1:L PR[91] 10mm/sec CNT100;
   1:  PR[GP1:91,1] = PR[GP1:90,1] + -7.783;
   1:  PR[GP1:91,2] = PR[GP1:90,2] + -19.535;
   1:L PR[91] 10mm/sec CNT100;
   1:  PR[GP1:91,1] = PR[GP1:90,1] + -6.682;
   1:  PR[GP1:91,2] = PR[GP1:90,2] + -19.495;
   1:L PR[91] 10mm/sec CNT100;
   1:  PR[GP1:91,1] = PR[GP1:90,1] + -6.365;
   1:  PR[GP1:91,2] = PR[GP1:90,2] + -19.449;
   1:L PR[91] 10mm/sec CNT100;
   1:  PR[GP1:91,1] = PR[GP1:90,1] + -3.225;
   1:  PR[GP1:91,2] = PR[GP1:90,2] + -18.895;
   1:L PR[91] 10mm/sec CNT100;
   1:  PR[GP1:91,1] = PR[GP1:90,1] + -1.064;
   1:  PR[GP1:91,2] = PR[GP1:90,2] + -18.175;
   1:L PR[91] 10mm/sec CNT100;
   1:  PR[GP1:91,1] = PR[GP1:90,1] + -0.528;
   1:  PR[GP1:91,2] = PR[GP1:90,2] + -17.959;
   1:L PR[91] 10mm/sec CNT100;
   1:  PR[GP1:91,1] = PR[GP1:90,1] + 0.147;
   1:  PR[GP1:91,2] = PR[GP1:90,2] + -17.652;
   1:L PR[91] 10mm/sec CNT100;
   1:  PR[GP1:91,1] = PR[GP1:90,1] + 0.981;
   1:  PR[GP1:91,2] = PR[GP1:90,2] + -17.447;
   1:L PR[91] 10mm/sec CNT100;
   1:  PR[GP1:91,1] = PR[GP1:90,1] + 2.340;
   1:  PR[GP1:91,2] = PR[GP1:90,2] + -17.791;
   1:L PR[91] 10mm/sec CNT100;
   1:  PR[GP1:91,1] = PR[GP1:90,1] + 3.506;
   1:  PR[GP1:91,2] = PR[GP1:90,2] + -18.381;
   1:L PR[91] 10mm/sec CNT100;
   1:  PR[GP1:91,1] = PR[GP1:90,1] + 4.099;
   1:  PR[GP1:91,2] = PR[GP1:90,2] + -18.655;
   1:L PR[91] 10mm/sec CNT100;
   1:  PR[GP1:91,1] = PR[GP1:90,1] + 6.735;
   1:  PR[GP1:91,2] = PR[GP1:90,2] + -19.548;
   1:L PR[91] 10mm/sec CNT100;
   1:  PR[GP1:91,1] = PR[GP1:90,1] + 9.498;
   1:  PR[GP1:91,2] = PR[GP1:90,2] + -20.000;
   1:L PR[91] 10mm/sec CNT100;
   1:  PR[GP1:91,1] = PR[GP1:90,1] + 12.267;
   1:  PR[GP1:91,2] = PR[GP1:90,2] + -20.016;
   1:L PR[91] 10mm/sec CNT100;
   1:  PR[GP1:91,1] = PR[GP1:90,1] + 12.509;
   1:  PR[GP1:91,2] = PR[GP1:90,2] + -19.994;
   1:L PR[91] 10mm/sec CNT100;
   1:  PR[GP1:91,1] = PR[GP1:90,1] + 14.866;
   1:  PR[GP1:91,2] = PR[GP1:90,2] + -19.655;
   1:L PR[91] 10mm/sec CNT100;
   1:  PR[GP1:91,1] = PR[GP1:90,1] + 15.733;
   1:  PR[GP1:91,2] = PR[GP1:90,2] + -19.449;
   1:L PR[91] 10mm/sec CNT100;
   1:  PR[GP1:91,1] = PR[GP1:90,1] + 17.304;
   1:  PR[GP1:91,2] = PR[GP1:90,2] + -18.973;
   1:L PR[91] 10mm/sec CNT100;
   1:  PR[GP1:91,1] = PR[GP1:90,1] + 18.826;
   1:  PR[GP1:91,2] = PR[GP1:90,2] + -18.370;
   1:L PR[91] 10mm/sec CNT100;
   1:  PR[GP1:91,1] = PR[GP1:90,1] + 19.542;
   1:  PR[GP1:91,2] = PR[GP1:90,2] + -18.030;
   1:L PR[91] 10mm/sec CNT100;
   1:  PR[GP1:91,1] = PR[GP1:90,1] + 21.622;
   1:  PR[GP1:91,2] = PR[GP1:90,2] + -16.849;
   1:L PR[91] 10mm/sec CNT100;
   1:  PR[GP1:91,1] = PR[GP1:90,1] + 23.835;
   1:  PR[GP1:91,2] = PR[GP1:90,2] + -15.246;
   1:L PR[91] 10mm/sec CNT100;
   1:  PR[GP1:91,1] = PR[GP1:90,1] + 24.722;
   1:  PR[GP1:91,2] = PR[GP1:90,2] + -14.405;
   1:L PR[91] 10mm/sec CNT100;
   1:  PR[GP1:91,1] = PR[GP1:90,1] + 25.801;
   1:  PR[GP1:91,2] = PR[GP1:90,2] + -13.363;
   1:L PR[91] 10mm/sec CNT100;
   1:  PR[GP1:91,1] = PR[GP1:90,1] + 27.483;
   1:  PR[GP1:91,2] = PR[GP1:90,2] + -11.221;
   1:L PR[91] 10mm/sec CNT100;
   1:  PR[GP1:91,1] = PR[GP1:90,1] + 28.127;
   1:  PR[GP1:91,2] = PR[GP1:90,2] + -10.099;
   1:L PR[91] 10mm/sec CNT100;
   1:  PR[GP1:91,1] = PR[GP1:90,1] + 28.862;
   1:  PR[GP1:91,2] = PR[GP1:90,2] + -8.876;
   1:L PR[91] 10mm/sec CNT100;
   1:  PR[GP1:91,1] = PR[GP1:90,1] + 29.885;
   1:  PR[GP1:91,2] = PR[GP1:90,2] + -6.394;
   1:L PR[91] 10mm/sec CNT100;
   1:  PR[GP1:91,1] = PR[GP1:90,1] + 30.506;
   1:  PR[GP1:91,2] = PR[GP1:90,2] + -3.808;
   1:L PR[91] 10mm/sec CNT100;
   1:  PR[GP1:91,1] = PR[GP1:90,1] + 30.600;
   1:  PR[GP1:91,2] = PR[GP1:90,2] + -2.486;
   1:L PR[91] 10mm/sec CNT100;
   1:  PR[GP1:91,1] = PR[GP1:90,1] + 30.672;
   1:  PR[GP1:91,2] = PR[GP1:90,2] + -1.170;
   1:L PR[91] 10mm/sec CNT100;
   1:  PR[GP1:91,1] = PR[GP1:90,1] + 30.277;
   1:  PR[GP1:91,2] = PR[GP1:90,2] + 2.205;
   1:L PR[91] 10mm/sec CNT100;
   1:  PR[GP1:91,1] = PR[GP1:90,1] + 29.186;
   1:  PR[GP1:91,2] = PR[GP1:90,2] + 5.399;
   1:L PR[91] 10mm/sec CNT100;
   1:  PR[GP1:91,1] = PR[GP1:90,1] + 27.422;
   1:  PR[GP1:91,2] = PR[GP1:90,2] + 8.308;
   1:L PR[91] 10mm/sec CNT100;
   1:  PR[GP1:91,1] = PR[GP1:90,1] + 25.079;
   1:  PR[GP1:91,2] = PR[GP1:90,2] + 10.806;
   1:L PR[91] 10mm/sec CNT100;
   1:  PR[GP1:91,1] = PR[GP1:90,1] + 22.253;
   1:  PR[GP1:91,2] = PR[GP1:90,2] + 12.801;
   1:L PR[91] 10mm/sec CNT100;
   1:  PR[GP1:91,1] = PR[GP1:90,1] + 19.033;
   1:  PR[GP1:91,2] = PR[GP1:90,2] + 14.232;
   1:L PR[91] 10mm/sec CNT100;
   1:  PR[GP1:91,1] = PR[GP1:90,1] + 15.573;
   1:  PR[GP1:91,2] = PR[GP1:90,2] + 15.034;
   1:L PR[91] 10mm/sec CNT100;
   1:  PR[GP1:91,1] = PR[GP1:90,1] + 12.011;
   1:  PR[GP1:91,2] = PR[GP1:90,2] + 15.180;
   1:L PR[91] 10mm/sec CNT100;
   1:  PR[GP1:91,1] = PR[GP1:90,1] + 8.467;
   1:  PR[GP1:91,2] = PR[GP1:90,2] + 14.671;
   1:L PR[91] 10mm/sec CNT100;
   1:  PR[GP1:91,1] = PR[GP1:90,1] + 5.077;
   1:  PR[GP1:91,2] = PR[GP1:90,2] + 13.530;
   1:L PR[91] 10mm/sec CNT100;
   1:  PR[GP1:91,1] = PR[GP1:90,1] + 1.991;
   1:  PR[GP1:91,2] = PR[GP1:90,2] + 11.780;
   1:L PR[91] 10mm/sec CNT100;
   1:  PR[GP1:91,1] = PR[GP1:90,1] + 1.747;
   1:  PR[GP1:91,2] = PR[GP1:90,2] + 11.627;
   1:L PR[91] 10mm/sec CNT100;
   1:  PR[GP1:91,1] = PR[GP1:90,1] + 1.385;
   1:  PR[GP1:91,2] = PR[GP1:90,2] + 11.355;
   1:L PR[91] 10mm/sec CNT100;
   1:  PR[GP1:91,1] = PR[GP1:90,1] + 0.642;
   1:  PR[GP1:91,2] = PR[GP1:90,2] + 11.051;
   1:L PR[91] 10mm/sec CNT100;
   1:  PR[GP1:91,1] = PR[GP1:90,1] + 0.360;
   1:  PR[GP1:91,2] = PR[GP1:90,2] + 10.896;
   1:L PR[91] 10mm/sec CNT100;
   1:  PR[GP1:91,1] = PR[GP1:90,1] + 0.042;
   1:  PR[GP1:91,2] = PR[GP1:90,2] + 10.859;
   1:L PR[91] 10mm/sec CNT100;
   1:  PR[GP1:91,1] = PR[GP1:90,1] + -0.658;
   1:  PR[GP1:91,2] = PR[GP1:90,2] + 10.957;
   1:L PR[91] 10mm/sec CNT100;
   1:  PR[GP1:91,1] = PR[GP1:90,1] + -0.977;
   1:  PR[GP1:91,2] = PR[GP1:90,2] + 10.963;
   1:L PR[91] 10mm/sec CNT100;
   1:  PR[GP1:91,1] = PR[GP1:90,1] + -1.474;
   1:  PR[GP1:91,2] = PR[GP1:90,2] + 11.211;
   1:L PR[91] 10mm/sec CNT100;
   1:  PR[GP1:91,1] = PR[GP1:90,1] + -2.253;
   1:  PR[GP1:91,2] = PR[GP1:90,2] + 11.681;
   1:L PR[91] 10mm/sec CNT100;
   1:  PR[GP1:91,1] = PR[GP1:90,1] + -3.648;
   1:  PR[GP1:91,2] = PR[GP1:90,2] + 12.367;
   1:L PR[91] 10mm/sec CNT100;
   1:  PR[GP1:91,1] = PR[GP1:90,1] + -6.463;
   1:  PR[GP1:91,2] = PR[GP1:90,2] + 13.524;
   1:L PR[91] 10mm/sec CNT100;
   1:  PR[GP1:91,1] = PR[GP1:90,1] + -6.654;
   1:  PR[GP1:91,2] = PR[GP1:90,2] + 13.592;
   1:L PR[91] 10mm/sec CNT100;
   1:  PR[GP1:91,1] = PR[GP1:90,1] + -9.735;
   1:  PR[GP1:91,2] = PR[GP1:90,2] + 14.402;
   1:L PR[91] 10mm/sec CNT100;
   1:  PR[GP1:91,1] = PR[GP1:90,1] + -11.168;
   1:  PR[GP1:91,2] = PR[GP1:90,2] + 14.655;
   1:L PR[91] 10mm/sec CNT100;
   1:  PR[GP1:91,1] = PR[GP1:90,1] + -12.953;
   1:  PR[GP1:91,2] = PR[GP1:90,2] + 14.821;
   1:L PR[91] 10mm/sec CNT100;
   1:  PR[GP1:91,1] = PR[GP1:90,1] + -15.957;
   1:  PR[GP1:91,2] = PR[GP1:90,2] + 14.810;
   1:L PR[91] 10mm/sec CNT100;
   1:  PR[GP1:91,1] = PR[GP1:90,1] + -16.380;
   1:  PR[GP1:91,2] = PR[GP1:90,2] + 14.777;
   1:L PR[91] 10mm/sec CNT100;
   1:  PR[GP1:91,1] = PR[GP1:90,1] + -17.816;
   1:  PR[GP1:91,2] = PR[GP1:90,2] + 14.503;
   1:L PR[91] 10mm/sec CNT100;
   1:  PR[GP1:91,1] = PR[GP1:90,1] + -20.036;
   1:  PR[GP1:91,2] = PR[GP1:90,2] + 14.043;
   1:L PR[91] 10mm/sec CNT100;
   1:  PR[GP1:91,1] = PR[GP1:90,1] + -22.485;
   1:  PR[GP1:91,2] = PR[GP1:90,2] + 13.010;
   1:L PR[91] 10mm/sec CNT100;
   1:  PR[GP1:91,1] = PR[GP1:90,1] + -23.468;
   1:  PR[GP1:91,2] = PR[GP1:90,2] + 12.572;
   1:L PR[91] 10mm/sec CNT100;
   1:  PR[GP1:91,1] = PR[GP1:90,1] + -25.162;
   1:  PR[GP1:91,2] = PR[GP1:90,2] + 11.396;
   1:L PR[91] 10mm/sec CNT100;
   1:  PR[GP1:91,1] = PR[GP1:90,1] + -26.428;
   1:  PR[GP1:91,2] = PR[GP1:90,2] + 10.489;
   1:L PR[91] 10mm/sec CNT100;
   1:  PR[GP1:91,1] = PR[GP1:90,1] + -28.807;
   1:  PR[GP1:91,2] = PR[GP1:90,2] + 7.887;
   1:L PR[91] 10mm/sec CNT100;
   1:  PR[GP1:91,1] = PR[GP1:90,1] + -29.493;
   1:  PR[GP1:91,2] = PR[GP1:90,2] + 6.704;
   1:L PR[91] 10mm/sec CNT100;
   1:  PR[GP1:91,1] = PR[GP1:90,1] + -30.538;
   1:  PR[GP1:91,2] = PR[GP1:90,2] + 4.882;
   1:L PR[91] 10mm/sec CNT100;
   1:  PR[GP1:91,1] = PR[GP1:90,1] + -31.592;
   1:  PR[GP1:91,2] = PR[GP1:90,2] + 1.612;
   1:L PR[91] 10mm/sec CNT100;
   1:  PR[GP1:91,1] = PR[GP1:90,1] + -31.833;
   1:  PR[GP1:91,2] = PR[GP1:90,2] + -1.848;
   1:L PR[91] 10mm/sec CNT100;
   1:  PR[GP1:91,1] = PR[GP1:90,1] + -31.550;
   1:  PR[GP1:91,2] = PR[GP1:90,2] + -3.773;
   1:L PR[91] 10mm/sec CNT100;
   1:  PR[GP1:91,1] = PR[GP1:90,1] + -31.293;
   1:  PR[GP1:91,2] = PR[GP1:90,2] + -5.386;
   1:L PR[91] 10mm/sec CNT100;
   1:  PR[GP1:91,1] = PR[GP1:90,1] + -30.742;
   1:  PR[GP1:91,2] = PR[GP1:90,2] + -6.911;
   1:L PR[91] 10mm/sec CNT100;
   1:  PR[GP1:91,1] = PR[GP1:90,1] + -30.036;
   1:  PR[GP1:91,2] = PR[GP1:90,2] + -8.791;
   1:L PR[91] 10mm/sec CNT100;
   1:  PR[GP1:91,1] = PR[GP1:90,1] + -29.417;
   1:  PR[GP1:91,2] = PR[GP1:90,2] + -9.781;
   1:L PR[91] 10mm/sec CNT100;
   1:  PR[GP1:91,1] = PR[GP1:90,1] + -27.977;
   1:  PR[GP1:91,2] = PR[GP1:90,2] + -11.972;
   1:L PR[91] 10mm/sec CNT100;
   1:  PR[GP1:91,1] = PR[GP1:90,1] + -27.608;
   1:  PR[GP1:91,2] = PR[GP1:90,2] + -12.360;
   1:L PR[91] 10mm/sec CNT100;
   1:  PR[GP1:91,1] = PR[GP1:90,1] + -25.941;
   1:  PR[GP1:91,2] = PR[GP1:90,2] + -14.025;
   1:L PR[91] 10mm/sec CNT100;
   1:  PR[GP1:91,1] = PR[GP1:90,1] + -25.211;
   1:  PR[GP1:91,2] = PR[GP1:90,2] + -14.725;
   1:L PR[91] 10mm/sec CNT100;
   1:  PR[GP1:91,1] = PR[GP1:90,1] + -23.552;
   1:  PR[GP1:91,2] = PR[GP1:90,2] + -15.615;
   1:  PR[GP1:91,3] = PR[GP1:90,3] + 29.700;
   1:L PR[91] 10mm/sec CNT100;
   1:  PR[GP1:91,1] = PR[GP1:90,1] + -21.555;
   1:  PR[GP1:91,2] = PR[GP1:90,2] + -16.916;
   1:L PR[91] 10mm/sec CNT100;
   1:  PR[GP1:91,1] = PR[GP1:90,1] + -18.647;
   1:  PR[GP1:91,2] = PR[GP1:90,2] + -18.247;
   1:L PR[91] 10mm/sec CNT100;
   1:  PR[GP1:91,1] = PR[GP1:90,1] + -18.235;
   1:  PR[GP1:91,2] = PR[GP1:90,2] + -18.419;
   1:L PR[91] 10mm/sec CNT100;
   1:  PR[GP1:91,1] = PR[GP1:90,1] + -14.749;
   1:  PR[GP1:91,2] = PR[GP1:90,2] + -19.372;
   1:L PR[91] 10mm/sec CNT100;
   1:  PR[GP1:91,1] = PR[GP1:90,1] + -13.511;
   1:  PR[GP1:91,2] = PR[GP1:90,2] + -19.599;
   1:L PR[91] 10mm/sec CNT100;
   1:  PR[GP1:91,1] = PR[GP1:90,1] + -11.723;
   1:  PR[GP1:91,2] = PR[GP1:90,2] + -19.797;
   1:L PR[91] 10mm/sec CNT100;
   1:  PR[GP1:91,1] = PR[GP1:90,1] + -9.213;
   1:  PR[GP1:91,2] = PR[GP1:90,2] + -19.935;
   1:L PR[91] 10mm/sec CNT100;
   1:  PR[GP1:91,1] = PR[GP1:90,1] + -5.953;
   1:  PR[GP1:91,2] = PR[GP1:90,2] + -19.815;
   1:L PR[91] 10mm/sec CNT100;
   1:  PR[GP1:91,1] = PR[GP1:90,1] + -4.949;
   1:  PR[GP1:91,2] = PR[GP1:90,2] + -19.671;
   1:L PR[91] 10mm/sec CNT100;
   1:  PR[GP1:91,1] = PR[GP1:90,1] + -2.297;
   1:  PR[GP1:91,2] = PR[GP1:90,2] + -19.203;
   1:L PR[91] 10mm/sec CNT100;
   1:  PR[GP1:91,1] = PR[GP1:90,1] + -0.440;
   1:  PR[GP1:91,2] = PR[GP1:90,2] + -18.584;
   1:L PR[91] 10mm/sec CNT100;
   1:  PR[GP1:91,1] = PR[GP1:90,1] + 0.521;
   1:  PR[GP1:91,2] = PR[GP1:90,2] + -18.187;
   1:L PR[91] 10mm/sec CNT100;
   1:  PR[GP1:91,1] = PR[GP1:90,1] + 1.221;
   1:  PR[GP1:91,2] = PR[GP1:90,2] + -18.026;
   1:L PR[91] 10mm/sec CNT100;
   1:  PR[GP1:91,1] = PR[GP1:90,1] + 2.578;
   1:  PR[GP1:91,2] = PR[GP1:90,2] + -18.316;
   1:L PR[91] 10mm/sec CNT100;
   1:  PR[GP1:91,1] = PR[GP1:90,1] + 3.835;
   1:  PR[GP1:91,2] = PR[GP1:90,2] + -18.901;
   1:L PR[91] 10mm/sec CNT100;
   1:  PR[GP1:91,1] = PR[GP1:90,1] + 6.465;
   1:  PR[GP1:91,2] = PR[GP1:90,2] + -19.802;
   1:L PR[91] 10mm/sec CNT100;
   1:  PR[GP1:91,1] = PR[GP1:90,1] + 9.221;
   1:  PR[GP1:91,2] = PR[GP1:90,2] + -20.265;
   1:L PR[91] 10mm/sec CNT100;
   1:  PR[GP1:91,1] = PR[GP1:90,1] + 12.050;
   1:  PR[GP1:91,2] = PR[GP1:90,2] + -20.274;
   1:L PR[91] 10mm/sec CNT100;
   1:  PR[GP1:91,1] = PR[GP1:90,1] + 14.880;
   1:  PR[GP1:91,2] = PR[GP1:90,2] + -19.824;
   1:L PR[91] 10mm/sec CNT100;
   1:  PR[GP1:91,1] = PR[GP1:90,1] + 17.389;
   1:  PR[GP1:91,2] = PR[GP1:90,2] + -19.065;
   1:L PR[91] 10mm/sec CNT100;
   1:  PR[GP1:91,1] = PR[GP1:90,1] + 18.024;
   1:  PR[GP1:91,2] = PR[GP1:90,2] + -18.813;
   1:L PR[91] 10mm/sec CNT100;
   1:  PR[GP1:91,1] = PR[GP1:90,1] + 19.660;
   1:  PR[GP1:91,2] = PR[GP1:90,2] + -18.036;
   1:L PR[91] 10mm/sec CNT100;
   1:  PR[GP1:91,1] = PR[GP1:90,1] + 20.932;
   1:  PR[GP1:91,2] = PR[GP1:90,2] + -17.309;
   1:L PR[91] 10mm/sec CNT100;
   1:  PR[GP1:91,1] = PR[GP1:90,1] + 21.696;
   1:  PR[GP1:91,2] = PR[GP1:90,2] + -16.795;
   1:L PR[91] 10mm/sec CNT100;
   1:  PR[GP1:91,1] = PR[GP1:90,1] + 23.483;
   1:  PR[GP1:91,2] = PR[GP1:90,2] + -15.407;
   1:L PR[91] 10mm/sec CNT100;
   1:  PR[GP1:91,1] = PR[GP1:90,1] + 25.458;
   1:  PR[GP1:91,2] = PR[GP1:90,2] + -13.494;
   1:L PR[91] 10mm/sec CNT100;
   1:  PR[GP1:91,1] = PR[GP1:90,1] + 27.125;
   1:  PR[GP1:91,2] = PR[GP1:90,2] + -11.356;
   1:L PR[91] 10mm/sec CNT100;
   1:  PR[GP1:91,1] = PR[GP1:90,1] + 28.465;
   1:  PR[GP1:91,2] = PR[GP1:90,2] + -9.010;
   1:L PR[91] 10mm/sec CNT100;
   1:  PR[GP1:91,1] = PR[GP1:90,1] + 29.447;
   1:  PR[GP1:91,2] = PR[GP1:90,2] + -6.503;
   1:L PR[91] 10mm/sec CNT100;
   1:  PR[GP1:91,1] = PR[GP1:90,1] + 30.061;
   1:  PR[GP1:91,2] = PR[GP1:90,2] + -3.926;
   1:L PR[91] 10mm/sec CNT100;
   1:  PR[GP1:91,1] = PR[GP1:90,1] + 30.231;
   1:  PR[GP1:91,2] = PR[GP1:90,2] + -1.305;
   1:L PR[91] 10mm/sec CNT100;
   1:  PR[GP1:91,1] = PR[GP1:90,1] + 29.829;
   1:  PR[GP1:91,2] = PR[GP1:90,2] + 2.083;
   1:L PR[91] 10mm/sec CNT100;
   1:  PR[GP1:91,1] = PR[GP1:90,1] + 28.736;
   1:  PR[GP1:91,2] = PR[GP1:90,2] + 5.282;
   1:L PR[91] 10mm/sec CNT100;
   1:  PR[GP1:91,1] = PR[GP1:90,1] + 26.985;
   1:  PR[GP1:91,2] = PR[GP1:90,2] + 8.180;
   1:L PR[91] 10mm/sec CNT100;
   1:  PR[GP1:91,1] = PR[GP1:90,1] + 24.649;
   1:  PR[GP1:91,2] = PR[GP1:90,2] + 10.674;
   1:L PR[91] 10mm/sec CNT100;
   1:  PR[GP1:91,1] = PR[GP1:90,1] + 21.817;
   1:  PR[GP1:91,2] = PR[GP1:90,2] + 12.673;
   1:L PR[91] 10mm/sec CNT100;
   1:  PR[GP1:91,1] = PR[GP1:90,1] + 18.591;
   1:  PR[GP1:91,2] = PR[GP1:90,2] + 14.108;
   1:L PR[91] 10mm/sec CNT100;
   1:  PR[GP1:91,1] = PR[GP1:90,1] + 15.187;
   1:  PR[GP1:91,2] = PR[GP1:90,2] + 14.888;
   1:L PR[91] 10mm/sec CNT100;
   1:  PR[GP1:91,1] = PR[GP1:90,1] + 13.327;
   1:  PR[GP1:91,2] = PR[GP1:90,2] + 14.966;
   1:L PR[91] 10mm/sec CNT100;
   1:  PR[GP1:91,1] = PR[GP1:90,1] + 11.650;
   1:  PR[GP1:91,2] = PR[GP1:90,2] + 15.029;
   1:L PR[91] 10mm/sec CNT100;
   1:  PR[GP1:91,1] = PR[GP1:90,1] + 8.101;
   1:  PR[GP1:91,2] = PR[GP1:90,2] + 14.526;
   1:L PR[91] 10mm/sec CNT100;
   1:  PR[GP1:91,1] = PR[GP1:90,1] + 4.769;
   1:  PR[GP1:91,2] = PR[GP1:90,2] + 13.369;
   1:L PR[91] 10mm/sec CNT100;
   1:  PR[GP1:91,1] = PR[GP1:90,1] + 4.056;
   1:  PR[GP1:91,2] = PR[GP1:90,2] + 12.998;
   1:L PR[91] 10mm/sec CNT100;
   1:  PR[GP1:91,1] = PR[GP1:90,1] + 1.470;
   1:  PR[GP1:91,2] = PR[GP1:90,2] + 11.531;
   1:L PR[91] 10mm/sec CNT100;
   1:  PR[GP1:91,1] = PR[GP1:90,1] + 0.407;
   1:  PR[GP1:91,2] = PR[GP1:90,2] + 11.115;
   1:L PR[91] 10mm/sec CNT100;
   1:  PR[GP1:91,1] = PR[GP1:90,1] + 0.117;
   1:  PR[GP1:91,2] = PR[GP1:90,2] + 11.086;
   1:L PR[91] 10mm/sec CNT100;
   1:  PR[GP1:91,1] = PR[GP1:90,1] + -0.907;
   1:  PR[GP1:91,2] = PR[GP1:90,2] + 11.244;
   1:L PR[91] 10mm/sec CNT100;
   1:  PR[GP1:91,1] = PR[GP1:90,1] + -1.357;
   1:  PR[GP1:91,2] = PR[GP1:90,2] + 11.447;
   1:L PR[91] 10mm/sec CNT100;
   1:  PR[GP1:91,1] = PR[GP1:90,1] + -3.299;
   1:  PR[GP1:91,2] = PR[GP1:90,2] + 12.401;
   1:L PR[91] 10mm/sec CNT100;
   1:  PR[GP1:91,1] = PR[GP1:90,1] + -4.889;
   1:  PR[GP1:91,2] = PR[GP1:90,2] + 13.055;
   1:L PR[91] 10mm/sec CNT100;
   1:  PR[GP1:91,1] = PR[GP1:90,1] + -6.081;
   1:  PR[GP1:91,2] = PR[GP1:90,2] + 13.481;
   1:L PR[91] 10mm/sec CNT100;
   1:  PR[GP1:91,1] = PR[GP1:90,1] + -8.673;
   1:  PR[GP1:91,2] = PR[GP1:90,2] + 14.109;
   1:L PR[91] 10mm/sec CNT100;
   1:  PR[GP1:91,1] = PR[GP1:90,1] + -9.570;
   1:  PR[GP1:91,2] = PR[GP1:90,2] + 14.348;
   1:L PR[91] 10mm/sec CNT100;
   1:  PR[GP1:91,1] = PR[GP1:90,1] + -10.030;
   1:  PR[GP1:91,2] = PR[GP1:90,2] + 14.430;
   1:L PR[91] 10mm/sec CNT100;
   1:  PR[GP1:91,1] = PR[GP1:90,1] + -12.732;
   1:  PR[GP1:91,2] = PR[GP1:90,2] + 14.681;
   1:L PR[91] 10mm/sec CNT100;
   1:  PR[GP1:91,1] = PR[GP1:90,1] + -14.796;
   1:  PR[GP1:91,2] = PR[GP1:90,2] + 14.673;
   1:L PR[91] 10mm/sec CNT100;
   1:  PR[GP1:91,1] = PR[GP1:90,1] + -16.095;
   1:  PR[GP1:91,2] = PR[GP1:90,2] + 14.570;
   1:L PR[91] 10mm/sec CNT100;
   1:  PR[GP1:91,1] = PR[GP1:90,1] + -19.414;
   1:  PR[GP1:91,2] = PR[GP1:90,2] + 13.939;
   1:L PR[91] 10mm/sec CNT100;
   1:  PR[GP1:91,1] = PR[GP1:90,1] + -19.528;
   1:  PR[GP1:91,2] = PR[GP1:90,2] + 13.909;
   1:L PR[91] 10mm/sec CNT100;
   1:  PR[GP1:91,1] = PR[GP1:90,1] + -20.129;
   1:  PR[GP1:91,2] = PR[GP1:90,2] + 13.669;
   1:L PR[91] 10mm/sec CNT100;
   1:  PR[GP1:91,1] = PR[GP1:90,1] + -22.958;
   1:  PR[GP1:91,2] = PR[GP1:90,2] + 12.463;
   1:L PR[91] 10mm/sec CNT100;
   1:  PR[GP1:91,1] = PR[GP1:90,1] + -25.133;
   1:  PR[GP1:91,2] = PR[GP1:90,2] + 10.954;
   1:L PR[91] 10mm/sec CNT100;
   1:  PR[GP1:91,1] = PR[GP1:90,1] + -25.934;
   1:  PR[GP1:91,2] = PR[GP1:90,2] + 10.380;
   1:L PR[91] 10mm/sec CNT100;
   1:  PR[GP1:91,1] = PR[GP1:90,1] + -28.327;
   1:  PR[GP1:91,2] = PR[GP1:90,2] + 7.770;
   1:L PR[91] 10mm/sec CNT100;
   1:  PR[GP1:91,1] = PR[GP1:90,1] + -30.068;
   1:  PR[GP1:91,2] = PR[GP1:90,2] + 4.753;
   1:L PR[91] 10mm/sec CNT100;
   1:  PR[GP1:91,1] = PR[GP1:90,1] + -31.128;
   1:  PR[GP1:91,2] = PR[GP1:90,2] + 1.473;
   1:L PR[91] 10mm/sec CNT100;
   1:  PR[GP1:91,1] = PR[GP1:90,1] + -31.367;
   1:  PR[GP1:91,2] = PR[GP1:90,2] + -2.002;
   1:L PR[91] 10mm/sec CNT100;
   1:  PR[GP1:91,1] = PR[GP1:90,1] + -31.166;
   1:  PR[GP1:91,2] = PR[GP1:90,2] + -3.368;
   1:L PR[91] 10mm/sec CNT100;
   1:  PR[GP1:91,1] = PR[GP1:90,1] + -30.816;
   1:  PR[GP1:91,2] = PR[GP1:90,2] + -5.557;
   1:L PR[91] 10mm/sec CNT100;
   1:  PR[GP1:91,1] = PR[GP1:90,1] + -29.546;
   1:  PR[GP1:91,2] = PR[GP1:90,2] + -8.982;
   1:L PR[91] 10mm/sec CNT100;
   1:  PR[GP1:91,1] = PR[GP1:90,1] + -29.239;
   1:  PR[GP1:91,2] = PR[GP1:90,2] + -9.472;
   1:L PR[91] 10mm/sec CNT100;
   1:  PR[GP1:91,1] = PR[GP1:90,1] + -27.470;
   1:  PR[GP1:91,2] = PR[GP1:90,2] + -12.160;
   1:L PR[91] 10mm/sec CNT100;
   1:  PR[GP1:91,1] = PR[GP1:90,1] + -24.695;
   1:  PR[GP1:91,2] = PR[GP1:90,2] + -14.824;
   1:L PR[91] 10mm/sec CNT100;
   1:  PR[GP1:91,1] = PR[GP1:90,1] + -22.158;
   1:  PR[GP1:91,2] = PR[GP1:90,2] + -16.322;
   1:  PR[GP1:91,3] = PR[GP1:90,3] + 30.800;
   1:L PR[91] 10mm/sec CNT100;
   1:  PR[GP1:91,1] = PR[GP1:90,1] + -21.098;
   1:  PR[GP1:91,2] = PR[GP1:90,2] + -17.012;
   1:L PR[91] 10mm/sec CNT100;
   1:  PR[GP1:91,1] = PR[GP1:90,1] + -17.703;
   1:  PR[GP1:91,2] = PR[GP1:90,2] + -18.561;
   1:L PR[91] 10mm/sec CNT100;
   1:  PR[GP1:91,1] = PR[GP1:90,1] + -17.149;
   1:  PR[GP1:91,2] = PR[GP1:90,2] + -18.739;
   1:L PR[91] 10mm/sec CNT100;
   1:  PR[GP1:91,1] = PR[GP1:90,1] + -14.339;
   1:  PR[GP1:91,2] = PR[GP1:90,2] + -19.516;
   1:L PR[91] 10mm/sec CNT100;
   1:  PR[GP1:91,1] = PR[GP1:90,1] + -12.174;
   1:  PR[GP1:91,2] = PR[GP1:90,2] + -19.913;
   1:L PR[91] 10mm/sec CNT100;
   1:  PR[GP1:91,1] = PR[GP1:90,1] + -11.486;
   1:  PR[GP1:91,2] = PR[GP1:90,2] + -19.990;
   1:L PR[91] 10mm/sec CNT100;
   1:  PR[GP1:91,1] = PR[GP1:90,1] + -10.451;
   1:  PR[GP1:91,2] = PR[GP1:90,2] + -20.047;
   1:L PR[91] 10mm/sec CNT100;
   1:  PR[GP1:91,1] = PR[GP1:90,1] + -8.607;
   1:  PR[GP1:91,2] = PR[GP1:90,2] + -20.209;
   1:L PR[91] 10mm/sec CNT100;
   1:  PR[GP1:91,1] = PR[GP1:90,1] + -8.054;
   1:  PR[GP1:91,2] = PR[GP1:90,2] + -20.238;
   1:L PR[91] 10mm/sec CNT100;
   1:  PR[GP1:91,1] = PR[GP1:90,1] + -5.223;
   1:  PR[GP1:91,2] = PR[GP1:90,2] + -20.135;
   1:L PR[91] 10mm/sec CNT100;
   1:  PR[GP1:91,1] = PR[GP1:90,1] + -3.532;
   1:  PR[GP1:91,2] = PR[GP1:90,2] + -19.893;
   1:L PR[91] 10mm/sec CNT100;
   1:  PR[GP1:91,1] = PR[GP1:90,1] + -1.370;
   1:  PR[GP1:91,2] = PR[GP1:90,2] + -19.512;
   1:L PR[91] 10mm/sec CNT100;
   1:  PR[GP1:91,1] = PR[GP1:90,1] + 0.190;
   1:  PR[GP1:91,2] = PR[GP1:90,2] + -18.990;
   1:L PR[91] 10mm/sec CNT100;
   1:  PR[GP1:91,1] = PR[GP1:90,1] + 0.895;
   1:  PR[GP1:91,2] = PR[GP1:90,2] + -18.711;
   1:L PR[91] 10mm/sec CNT100;
   1:  PR[GP1:91,1] = PR[GP1:90,1] + 1.488;
   1:  PR[GP1:91,2] = PR[GP1:90,2] + -18.569;
   1:L PR[91] 10mm/sec CNT100;
   1:  PR[GP1:91,1] = PR[GP1:90,1] + 2.847;
   1:  PR[GP1:91,2] = PR[GP1:90,2] + -18.823;
   1:L PR[91] 10mm/sec CNT100;
   1:  PR[GP1:91,1] = PR[GP1:90,1] + 3.566;
   1:  PR[GP1:91,2] = PR[GP1:90,2] + -19.145;
   1:L PR[91] 10mm/sec CNT100;
   1:  PR[GP1:91,1] = PR[GP1:90,1] + 6.194;
   1:  PR[GP1:91,2] = PR[GP1:90,2] + -20.056;
   1:L PR[91] 10mm/sec CNT100;
   1:  PR[GP1:91,1] = PR[GP1:90,1] + 8.944;
   1:  PR[GP1:91,2] = PR[GP1:90,2] + -20.529;
   1:L PR[91] 10mm/sec CNT100;
   1:  PR[GP1:91,1] = PR[GP1:90,1] + 10.270;
   1:  PR[GP1:91,2] = PR[GP1:90,2] + -20.530;
   1:L PR[91] 10mm/sec CNT100;
   1:  PR[GP1:91,1] = PR[GP1:90,1] + 11.775;
   1:  PR[GP1:91,2] = PR[GP1:90,2] + -20.551;
   1:L PR[91] 10mm/sec CNT100;
   1:  PR[GP1:91,1] = PR[GP1:90,1] + 14.600;
   1:  PR[GP1:91,2] = PR[GP1:90,2] + -20.114;
   1:L PR[91] 10mm/sec CNT100;
   1:  PR[GP1:91,1] = PR[GP1:90,1] + 17.353;
   1:  PR[GP1:91,2] = PR[GP1:90,2] + -19.219;
   1:L PR[91] 10mm/sec CNT100;
   1:  PR[GP1:91,1] = PR[GP1:90,1] + 18.110;
   1:  PR[GP1:91,2] = PR[GP1:90,2] + -18.835;
   1:L PR[91] 10mm/sec CNT100;
   1:  PR[GP1:91,1] = PR[GP1:90,1] + 19.778;
   1:  PR[GP1:91,2] = PR[GP1:90,2] + -18.042;
   1:L PR[91] 10mm/sec CNT100;
   1:  PR[GP1:91,1] = PR[GP1:90,1] + 20.205;
   1:  PR[GP1:91,2] = PR[GP1:90,2] + -17.798;
   1:L PR[91] 10mm/sec CNT100;
   1:  PR[GP1:91,1] = PR[GP1:90,1] + 21.831;
   1:  PR[GP1:91,2] = PR[GP1:90,2] + -16.703;
   1:L PR[91] 10mm/sec CNT100;
   1:  PR[GP1:91,1] = PR[GP1:90,1] + 22.848;
   1:  PR[GP1:91,2] = PR[GP1:90,2] + -15.913;
   1:L PR[91] 10mm/sec CNT100;
   1:  PR[GP1:91,1] = PR[GP1:90,1] + 23.627;
   1:  PR[GP1:91,2] = PR[GP1:90,2] + -15.198;
   1:L PR[91] 10mm/sec CNT100;
   1:  PR[GP1:91,1] = PR[GP1:90,1] + 25.060;
   1:  PR[GP1:91,2] = PR[GP1:90,2] + -13.719;
   1:L PR[91] 10mm/sec CNT100;
   1:  PR[GP1:91,1] = PR[GP1:90,1] + 25.553;
   1:  PR[GP1:91,2] = PR[GP1:90,2] + -13.056;
   1:L PR[91] 10mm/sec CNT100;
   1:  PR[GP1:91,1] = PR[GP1:90,1] + 26.766;
   1:  PR[GP1:91,2] = PR[GP1:90,2] + -11.491;
   1:L PR[91] 10mm/sec CNT100;
   1:  PR[GP1:91,1] = PR[GP1:90,1] + 28.094;
   1:  PR[GP1:91,2] = PR[GP1:90,2] + -9.153;
   1:L PR[91] 10mm/sec CNT100;
   1:  PR[GP1:91,1] = PR[GP1:90,1] + 28.642;
   1:  PR[GP1:91,2] = PR[GP1:90,2] + -7.754;
   1:L PR[91] 10mm/sec CNT100;
   1:  PR[GP1:91,1] = PR[GP1:90,1] + 29.065;
   1:  PR[GP1:91,2] = PR[GP1:90,2] + -6.662;
   1:L PR[91] 10mm/sec CNT100;
   1:  PR[GP1:91,1] = PR[GP1:90,1] + 29.646;
   1:  PR[GP1:91,2] = PR[GP1:90,2] + -4.076;
   1:L PR[91] 10mm/sec CNT100;
   1:  PR[GP1:91,1] = PR[GP1:90,1] + 29.797;
   1:  PR[GP1:91,2] = PR[GP1:90,2] + -1.450;
   1:L PR[91] 10mm/sec CNT100;
   1:  PR[GP1:91,1] = PR[GP1:90,1] + 29.406;
   1:  PR[GP1:91,2] = PR[GP1:90,2] + 1.937;
   1:L PR[91] 10mm/sec CNT100;
   1:  PR[GP1:91,1] = PR[GP1:90,1] + 28.314;
   1:  PR[GP1:91,2] = PR[GP1:90,2] + 5.140;
   1:L PR[91] 10mm/sec CNT100;
   1:  PR[GP1:91,1] = PR[GP1:90,1] + 26.560;
   1:  PR[GP1:91,2] = PR[GP1:90,2] + 8.043;
   1:L PR[91] 10mm/sec CNT100;
   1:  PR[GP1:91,1] = PR[GP1:90,1] + 24.219;
   1:  PR[GP1:91,2] = PR[GP1:90,2] + 10.541;
   1:L PR[91] 10mm/sec CNT100;
   1:  PR[GP1:91,1] = PR[GP1:90,1] + 21.382;
   1:  PR[GP1:91,2] = PR[GP1:90,2] + 12.544;
   1:L PR[91] 10mm/sec CNT100;
   1:  PR[GP1:91,1] = PR[GP1:90,1] + 18.225;
   1:  PR[GP1:91,2] = PR[GP1:90,2] + 13.951;
   1:L PR[91] 10mm/sec CNT100;
   1:  PR[GP1:91,1] = PR[GP1:90,1] + 14.801;
   1:  PR[GP1:91,2] = PR[GP1:90,2] + 14.742;
   1:L PR[91] 10mm/sec CNT100;
   1:  PR[GP1:91,1] = PR[GP1:90,1] + 11.287;
   1:  PR[GP1:91,2] = PR[GP1:90,2] + 14.877;
   1:L PR[91] 10mm/sec CNT100;
   1:  PR[GP1:91,1] = PR[GP1:90,1] + 9.513;
   1:  PR[GP1:91,2] = PR[GP1:90,2] + 14.629;
   1:L PR[91] 10mm/sec CNT100;
   1:  PR[GP1:91,1] = PR[GP1:90,1] + 7.805;
   1:  PR[GP1:91,2] = PR[GP1:90,2] + 14.363;
   1:L PR[91] 10mm/sec CNT100;
   1:  PR[GP1:91,1] = PR[GP1:90,1] + 4.468;
   1:  PR[GP1:91,2] = PR[GP1:90,2] + 13.209;
   1:L PR[91] 10mm/sec CNT100;
   1:  PR[GP1:91,1] = PR[GP1:90,1] + 3.129;
   1:  PR[GP1:91,2] = PR[GP1:90,2] + 12.513;
   1:L PR[91] 10mm/sec CNT100;
   1:  PR[GP1:91,1] = PR[GP1:90,1] + 1.599;
   1:  PR[GP1:91,2] = PR[GP1:90,2] + 11.652;
   1:L PR[91] 10mm/sec CNT100;
   1:  PR[GP1:91,1] = PR[GP1:90,1] + 1.028;
   1:  PR[GP1:91,2] = PR[GP1:90,2] + 11.485;
   1:L PR[91] 10mm/sec CNT100;
   1:  PR[GP1:91,1] = PR[GP1:90,1] + 0.486;
   1:  PR[GP1:91,2] = PR[GP1:90,2] + 11.276;
   1:L PR[91] 10mm/sec CNT100;
   1:  PR[GP1:91,1] = PR[GP1:90,1] + 0.241;
   1:  PR[GP1:91,2] = PR[GP1:90,2] + 11.251;
   1:L PR[91] 10mm/sec CNT100;
   1:  PR[GP1:91,1] = PR[GP1:90,1] + -0.587;
   1:  PR[GP1:91,2] = PR[GP1:90,2] + 11.435;
   1:L PR[91] 10mm/sec CNT100;
   1:  PR[GP1:91,1] = PR[GP1:90,1] + -0.835;
   1:  PR[GP1:91,2] = PR[GP1:90,2] + 11.470;
   1:L PR[91] 10mm/sec CNT100;
   1:  PR[GP1:91,1] = PR[GP1:90,1] + -2.479;
   1:  PR[GP1:91,2] = PR[GP1:90,2] + 12.204;
   1:L PR[91] 10mm/sec CNT100;
   1:  PR[GP1:91,1] = PR[GP1:90,1] + -2.950;
   1:  PR[GP1:91,2] = PR[GP1:90,2] + 12.435;
   1:L PR[91] 10mm/sec CNT100;
   1:  PR[GP1:91,1] = PR[GP1:90,1] + -3.315;
   1:  PR[GP1:91,2] = PR[GP1:90,2] + 12.585;
   1:L PR[91] 10mm/sec CNT100;
   1:  PR[GP1:91,1] = PR[GP1:90,1] + -5.513;
   1:  PR[GP1:91,2] = PR[GP1:90,2] + 13.372;
   1:L PR[91] 10mm/sec CNT100;
   1:  PR[GP1:91,1] = PR[GP1:90,1] + -9.048;
   1:  PR[GP1:91,2] = PR[GP1:90,2] + 14.221;
   1:L PR[91] 10mm/sec CNT100;
   1:  PR[GP1:91,1] = PR[GP1:90,1] + -12.512;
   1:  PR[GP1:91,2] = PR[GP1:90,2] + 14.540;
   1:L PR[91] 10mm/sec CNT100;
   1:  PR[GP1:91,1] = PR[GP1:90,1] + -13.635;
   1:  PR[GP1:91,2] = PR[GP1:90,2] + 14.536;
   1:L PR[91] 10mm/sec CNT100;
   1:  PR[GP1:91,1] = PR[GP1:90,1] + -15.810;
   1:  PR[GP1:91,2] = PR[GP1:90,2] + 14.364;
   1:L PR[91] 10mm/sec CNT100;
   1:  PR[GP1:91,1] = PR[GP1:90,1] + -18.258;
   1:  PR[GP1:91,2] = PR[GP1:90,2] + 13.898;
   1:L PR[91] 10mm/sec CNT100;
   1:  PR[GP1:91,1] = PR[GP1:90,1] + -19.175;
   1:  PR[GP1:91,2] = PR[GP1:90,2] + 13.657;
   1:L PR[91] 10mm/sec CNT100;
   1:  PR[GP1:91,1] = PR[GP1:90,1] + -22.456;
   1:  PR[GP1:91,2] = PR[GP1:90,2] + 12.342;
   1:L PR[91] 10mm/sec CNT100;
   1:  PR[GP1:91,1] = PR[GP1:90,1] + -25.443;
   1:  PR[GP1:91,2] = PR[GP1:90,2] + 10.268;
   1:L PR[91] 10mm/sec CNT100;
   1:  PR[GP1:91,1] = PR[GP1:90,1] + -27.847;
   1:  PR[GP1:91,2] = PR[GP1:90,2] + 7.653;
   1:L PR[91] 10mm/sec CNT100;
   1:  PR[GP1:91,1] = PR[GP1:90,1] + -29.597;
   1:  PR[GP1:91,2] = PR[GP1:90,2] + 4.625;
   1:L PR[91] 10mm/sec CNT100;
   1:  PR[GP1:91,1] = PR[GP1:90,1] + -30.664;
   1:  PR[GP1:91,2] = PR[GP1:90,2] + 1.333;
   1:L PR[91] 10mm/sec CNT100;
   1:  PR[GP1:91,1] = PR[GP1:90,1] + -30.900;
   1:  PR[GP1:91,2] = PR[GP1:90,2] + -2.153;
   1:L PR[91] 10mm/sec CNT100;
   1:  PR[GP1:91,1] = PR[GP1:90,1] + -30.339;
   1:  PR[GP1:91,2] = PR[GP1:90,2] + -5.731;
   1:L PR[91] 10mm/sec CNT100;
   1:  PR[GP1:91,1] = PR[GP1:90,1] + -29.057;
   1:  PR[GP1:91,2] = PR[GP1:90,2] + -9.168;
   1:L PR[91] 10mm/sec CNT100;
   1:  PR[GP1:91,1] = PR[GP1:90,1] + -26.908;
   1:  PR[GP1:91,2] = PR[GP1:90,2] + -12.275;
   1:L PR[91] 10mm/sec CNT100;
   1:  PR[GP1:91,1] = PR[GP1:90,1] + -26.246;
   1:  PR[GP1:91,2] = PR[GP1:90,2] + -12.939;
   1:L PR[91] 10mm/sec CNT100;
   1:  PR[GP1:91,1] = PR[GP1:90,1] + -24.178;
   1:  PR[GP1:91,2] = PR[GP1:90,2] + -14.923;
   1:L PR[91] 10mm/sec CNT100;
   1:  PR[GP1:91,1] = PR[GP1:90,1] + -20.764;
   1:  PR[GP1:91,2] = PR[GP1:90,2] + -17.028;
   1:  PR[GP1:91,3] = PR[GP1:90,3] + 31.900;
   1:L PR[91] 10mm/sec CNT100;
   1:  PR[GP1:91,1] = PR[GP1:90,1] + -20.640;
   1:  PR[GP1:91,2] = PR[GP1:90,2] + -17.108;
   1:L PR[91] 10mm/sec CNT100;
   1:  PR[GP1:91,1] = PR[GP1:90,1] + -17.113;
   1:  PR[GP1:91,2] = PR[GP1:90,2] + -18.711;
   1:L PR[91] 10mm/sec CNT100;
   1:  PR[GP1:91,1] = PR[GP1:90,1] + -15.525;
   1:  PR[GP1:91,2] = PR[GP1:90,2] + -19.219;
   1:L PR[91] 10mm/sec CNT100;
   1:  PR[GP1:91,1] = PR[GP1:90,1] + -13.929;
   1:  PR[GP1:91,2] = PR[GP1:90,2] + -19.661;
   1:L PR[91] 10mm/sec CNT100;
   1:  PR[GP1:91,1] = PR[GP1:90,1] + -11.684;
   1:  PR[GP1:91,2] = PR[GP1:90,2] + -20.073;
   1:L PR[91] 10mm/sec CNT100;
   1:  PR[GP1:91,1] = PR[GP1:90,1] + -10.976;
   1:  PR[GP1:91,2] = PR[GP1:90,2] + -20.224;
   1:L PR[91] 10mm/sec CNT100;
   1:  PR[GP1:91,1] = PR[GP1:90,1] + -8.054;
   1:  PR[GP1:91,2] = PR[GP1:90,2] + -20.482;
   1:L PR[91] 10mm/sec CNT100;
   1:  PR[GP1:91,1] = PR[GP1:90,1] + -6.893;
   1:  PR[GP1:91,2] = PR[GP1:90,2] + -20.543;
   1:L PR[91] 10mm/sec CNT100;
   1:  PR[GP1:91,1] = PR[GP1:90,1] + -4.494;
   1:  PR[GP1:91,2] = PR[GP1:90,2] + -20.456;
   1:L PR[91] 10mm/sec CNT100;
   1:  PR[GP1:91,1] = PR[GP1:90,1] + -2.116;
   1:  PR[GP1:91,2] = PR[GP1:90,2] + -20.115;
   1:L PR[91] 10mm/sec CNT100;
   1:  PR[GP1:91,1] = PR[GP1:90,1] + -0.443;
   1:  PR[GP1:91,2] = PR[GP1:90,2] + -19.820;
   1:L PR[91] 10mm/sec CNT100;
   1:  PR[GP1:91,1] = PR[GP1:90,1] + 0.820;
   1:  PR[GP1:91,2] = PR[GP1:90,2] + -19.397;
   1:L PR[91] 10mm/sec CNT100;
   1:  PR[GP1:91,1] = PR[GP1:90,1] + 1.289;
   1:  PR[GP1:91,2] = PR[GP1:90,2] + -19.219;
   1:L PR[91] 10mm/sec CNT100;
   1:  PR[GP1:91,1] = PR[GP1:90,1] + 1.768;
   1:  PR[GP1:91,2] = PR[GP1:90,2] + -19.106;
   1:L PR[91] 10mm/sec CNT100;
   1:  PR[GP1:91,1] = PR[GP1:90,1] + 3.109;
   1:  PR[GP1:91,2] = PR[GP1:90,2] + -19.314;
   1:L PR[91] 10mm/sec CNT100;
   1:  PR[GP1:91,1] = PR[GP1:90,1] + 5.925;
   1:  PR[GP1:91,2] = PR[GP1:90,2] + -20.310;
   1:L PR[91] 10mm/sec CNT100;
   1:  PR[GP1:91,1] = PR[GP1:90,1] + 8.672;
   1:  PR[GP1:91,2] = PR[GP1:90,2] + -20.794;
   1:L PR[91] 10mm/sec CNT100;
   1:  PR[GP1:91,1] = PR[GP1:90,1] + 11.496;
   1:  PR[GP1:91,2] = PR[GP1:90,2] + -20.828;
   1:L PR[91] 10mm/sec CNT100;
   1:  PR[GP1:91,1] = PR[GP1:90,1] + 14.322;
   1:  PR[GP1:91,2] = PR[GP1:90,2] + -20.405;
   1:L PR[91] 10mm/sec CNT100;
   1:  PR[GP1:91,1] = PR[GP1:90,1] + 17.075;
   1:  PR[GP1:91,2] = PR[GP1:90,2] + -19.526;
   1:L PR[91] 10mm/sec CNT100;
   1:  PR[GP1:91,1] = PR[GP1:90,1] + 19.683;
   1:  PR[GP1:91,2] = PR[GP1:90,2] + -18.210;
   1:L PR[91] 10mm/sec CNT100;
   1:  PR[GP1:91,1] = PR[GP1:90,1] + 21.021;
   1:  PR[GP1:91,2] = PR[GP1:90,2] + -17.247;
   1:L PR[91] 10mm/sec CNT100;
   1:  PR[GP1:91,1] = PR[GP1:90,1] + 21.966;
   1:  PR[GP1:91,2] = PR[GP1:90,2] + -16.611;
   1:L PR[91] 10mm/sec CNT100;
   1:  PR[GP1:91,1] = PR[GP1:90,1] + 22.205;
   1:  PR[GP1:91,2] = PR[GP1:90,2] + -16.425;
   1:L PR[91] 10mm/sec CNT100;
   1:  PR[GP1:91,1] = PR[GP1:90,1] + 23.758;
   1:  PR[GP1:91,2] = PR[GP1:90,2] + -15.002;
   1:L PR[91] 10mm/sec CNT100;
   1:  PR[GP1:91,1] = PR[GP1:90,1] + 24.515;
   1:  PR[GP1:91,2] = PR[GP1:90,2] + -14.219;
   1:L PR[91] 10mm/sec CNT100;
   1:  PR[GP1:91,1] = PR[GP1:90,1] + 25.282;
   1:  PR[GP1:91,2] = PR[GP1:90,2] + -13.267;
   1:L PR[91] 10mm/sec CNT100;
   1:  PR[GP1:91,1] = PR[GP1:90,1] + 26.356;
   1:  PR[GP1:91,2] = PR[GP1:90,2] + -11.784;
   1:L PR[91] 10mm/sec CNT100;
   1:  PR[GP1:91,1] = PR[GP1:90,1] + 26.558;
   1:  PR[GP1:91,2] = PR[GP1:90,2] + -11.436;
   1:L PR[91] 10mm/sec CNT100;
   1:  PR[GP1:91,1] = PR[GP1:90,1] + 27.217;
   1:  PR[GP1:91,2] = PR[GP1:90,2] + -10.189;
   1:L PR[91] 10mm/sec CNT100;
   1:  PR[GP1:91,1] = PR[GP1:90,1] + 27.722;
   1:  PR[GP1:91,2] = PR[GP1:90,2] + -9.296;
   1:L PR[91] 10mm/sec CNT100;
   1:  PR[GP1:91,1] = PR[GP1:90,1] + 28.684;
   1:  PR[GP1:91,2] = PR[GP1:90,2] + -6.816;
   1:L PR[91] 10mm/sec CNT100;
   1:  PR[GP1:91,1] = PR[GP1:90,1] + 29.260;
   1:  PR[GP1:91,2] = PR[GP1:90,2] + -4.244;
   1:L PR[91] 10mm/sec CNT100;
   1:  PR[GP1:91,1] = PR[GP1:90,1] + 29.400;
   1:  PR[GP1:91,2] = PR[GP1:90,2] + -1.628;
   1:L PR[91] 10mm/sec CNT100;
   1:  PR[GP1:91,1] = PR[GP1:90,1] + 28.985;
   1:  PR[GP1:91,2] = PR[GP1:90,2] + 1.788;
   1:L PR[91] 10mm/sec CNT100;
   1:  PR[GP1:91,1] = PR[GP1:90,1] + 27.893;
   1:  PR[GP1:91,2] = PR[GP1:90,2] + 4.998;
   1:L PR[91] 10mm/sec CNT100;
   1:  PR[GP1:91,1] = PR[GP1:90,1] + 26.135;
   1:  PR[GP1:91,2] = PR[GP1:90,2] + 7.906;
   1:L PR[91] 10mm/sec CNT100;
   1:  PR[GP1:91,1] = PR[GP1:90,1] + 23.791;
   1:  PR[GP1:91,2] = PR[GP1:90,2] + 10.409;
   1:L PR[91] 10mm/sec CNT100;
   1:  PR[GP1:91,1] = PR[GP1:90,1] + 21.014;
   1:  PR[GP1:91,2] = PR[GP1:90,2] + 12.385;
   1:L PR[91] 10mm/sec CNT100;
   1:  PR[GP1:91,1] = PR[GP1:90,1] + 17.860;
   1:  PR[GP1:91,2] = PR[GP1:90,2] + 13.793;
   1:L PR[91] 10mm/sec CNT100;
   1:  PR[GP1:91,1] = PR[GP1:90,1] + 14.421;
   1:  PR[GP1:91,2] = PR[GP1:90,2] + 14.594;
   1:L PR[91] 10mm/sec CNT100;
   1:  PR[GP1:91,1] = PR[GP1:90,1] + 10.931;
   1:  PR[GP1:91,2] = PR[GP1:90,2] + 14.726;
   1:L PR[91] 10mm/sec CNT100;
   1:  PR[GP1:91,1] = PR[GP1:90,1] + 7.505;
   1:  PR[GP1:91,2] = PR[GP1:90,2] + 14.199;
   1:L PR[91] 10mm/sec CNT100;
   1:  PR[GP1:91,1] = PR[GP1:90,1] + 4.168;
   1:  PR[GP1:91,2] = PR[GP1:90,2] + 13.049;
   1:L PR[91] 10mm/sec CNT100;
   1:  PR[GP1:91,1] = PR[GP1:90,1] + 2.203;
   1:  PR[GP1:91,2] = PR[GP1:90,2] + 12.027;
   1:L PR[91] 10mm/sec CNT100;
   1:  PR[GP1:91,1] = PR[GP1:90,1] + 1.759;
   1:  PR[GP1:91,2] = PR[GP1:90,2] + 11.778;
   1:L PR[91] 10mm/sec CNT100;
   1:  PR[GP1:91,1] = PR[GP1:90,1] + 0.458;
   1:  PR[GP1:91,2] = PR[GP1:90,2] + 11.392;
   1:L PR[91] 10mm/sec CNT100;
   1:  PR[GP1:91,1] = PR[GP1:90,1] + -0.674;
   1:  PR[GP1:91,2] = PR[GP1:90,2] + 11.631;
   1:L PR[91] 10mm/sec CNT100;
   1:  PR[GP1:91,1] = PR[GP1:90,1] + -1.696;
   1:  PR[GP1:91,2] = PR[GP1:90,2] + 12.087;
   1:L PR[91] 10mm/sec CNT100;
   1:  PR[GP1:91,1] = PR[GP1:90,1] + -2.280;
   1:  PR[GP1:91,2] = PR[GP1:90,2] + 12.329;
   1:L PR[91] 10mm/sec CNT100;
   1:  PR[GP1:91,1] = PR[GP1:90,1] + -4.945;
   1:  PR[GP1:91,2] = PR[GP1:90,2] + 13.263;
   1:L PR[91] 10mm/sec CNT100;
   1:  PR[GP1:91,1] = PR[GP1:90,1] + -6.229;
   1:  PR[GP1:91,2] = PR[GP1:90,2] + 13.574;
   1:L PR[91] 10mm/sec CNT100;
   1:  PR[GP1:91,1] = PR[GP1:90,1] + -8.202;
   1:  PR[GP1:91,2] = PR[GP1:90,2] + 14.029;
   1:L PR[91] 10mm/sec CNT100;
   1:  PR[GP1:91,1] = PR[GP1:90,1] + -9.043;
   1:  PR[GP1:91,2] = PR[GP1:90,2] + 14.126;
   1:L PR[91] 10mm/sec CNT100;
   1:  PR[GP1:91,1] = PR[GP1:90,1] + -12.288;
   1:  PR[GP1:91,2] = PR[GP1:90,2] + 14.400;
   1:L PR[91] 10mm/sec CNT100;
   1:  PR[GP1:91,1] = PR[GP1:90,1] + -12.474;
   1:  PR[GP1:91,2] = PR[GP1:90,2] + 14.399;
   1:L PR[91] 10mm/sec CNT100;
   1:  PR[GP1:91,1] = PR[GP1:90,1] + -15.526;
   1:  PR[GP1:91,2] = PR[GP1:90,2] + 14.158;
   1:L PR[91] 10mm/sec CNT100;
   1:  PR[GP1:91,1] = PR[GP1:90,1] + -17.103;
   1:  PR[GP1:91,2] = PR[GP1:90,2] + 13.858;
   1:L PR[91] 10mm/sec CNT100;
   1:  PR[GP1:91,1] = PR[GP1:90,1] + -18.823;
   1:  PR[GP1:91,2] = PR[GP1:90,2] + 13.404;
   1:L PR[91] 10mm/sec CNT100;
   1:  PR[GP1:91,1] = PR[GP1:90,1] + -21.336;
   1:  PR[GP1:91,2] = PR[GP1:90,2] + 12.400;
   1:L PR[91] 10mm/sec CNT100;
   1:  PR[GP1:91,1] = PR[GP1:90,1] + -22.025;
   1:  PR[GP1:91,2] = PR[GP1:90,2] + 12.072;
   1:L PR[91] 10mm/sec CNT100;
   1:  PR[GP1:91,1] = PR[GP1:90,1] + -24.961;
   1:  PR[GP1:91,2] = PR[GP1:90,2] + 10.123;
   1:L PR[91] 10mm/sec CNT100;
   1:  PR[GP1:91,1] = PR[GP1:90,1] + -25.490;
   1:  PR[GP1:91,2] = PR[GP1:90,2] + 9.573;
   1:L PR[91] 10mm/sec CNT100;
   1:  PR[GP1:91,1] = PR[GP1:90,1] + -27.367;
   1:  PR[GP1:91,2] = PR[GP1:90,2] + 7.536;
   1:L PR[91] 10mm/sec CNT100;
   1:  PR[GP1:91,1] = PR[GP1:90,1] + -29.126;
   1:  PR[GP1:91,2] = PR[GP1:90,2] + 4.497;
   1:L PR[91] 10mm/sec CNT100;
   1:  PR[GP1:91,1] = PR[GP1:90,1] + -30.200;
   1:  PR[GP1:91,2] = PR[GP1:90,2] + 1.194;
   1:L PR[91] 10mm/sec CNT100;
   1:  PR[GP1:91,1] = PR[GP1:90,1] + -30.433;
   1:  PR[GP1:91,2] = PR[GP1:90,2] + -2.307;
   1:L PR[91] 10mm/sec CNT100;
   1:  PR[GP1:91,1] = PR[GP1:90,1] + -29.875;
   1:  PR[GP1:91,2] = PR[GP1:90,2] + -5.828;
   1:L PR[91] 10mm/sec CNT100;
   1:  PR[GP1:91,1] = PR[GP1:90,1] + -29.864;
   1:  PR[GP1:91,2] = PR[GP1:90,2] + -5.887;
   1:L PR[91] 10mm/sec CNT100;
   1:  PR[GP1:91,1] = PR[GP1:90,1] + -28.479;
   1:  PR[GP1:91,2] = PR[GP1:90,2] + -9.298;
   1:L PR[91] 10mm/sec CNT100;
   1:  PR[GP1:91,1] = PR[GP1:90,1] + -28.082;
   1:  PR[GP1:91,2] = PR[GP1:90,2] + -9.889;
   1:L PR[91] 10mm/sec CNT100;
   1:  PR[GP1:91,1] = PR[GP1:90,1] + -26.345;
   1:  PR[GP1:91,2] = PR[GP1:90,2] + -12.389;
   1:L PR[91] 10mm/sec CNT100;
   1:  PR[GP1:91,1] = PR[GP1:90,1] + -24.989;
   1:  PR[GP1:91,2] = PR[GP1:90,2] + -13.748;
   1:L PR[91] 10mm/sec CNT100;
   1:  PR[GP1:91,1] = PR[GP1:90,1] + -23.662;
   1:  PR[GP1:91,2] = PR[GP1:90,2] + -15.022;
   1:L PR[91] 10mm/sec CNT100;
   1:  PR[GP1:91,1] = PR[GP1:90,1] + -23.145;
   1:  PR[GP1:91,2] = PR[GP1:90,2] + -15.120;
   1:  PR[GP1:91,3] = PR[GP1:90,3] + 33.000;
   1:L PR[91] 10mm/sec CNT100;
   1:  PR[GP1:91,1] = PR[GP1:90,1] + -21.606;
   1:  PR[GP1:91,2] = PR[GP1:90,2] + -16.186;
   1:L PR[91] 10mm/sec CNT100;
   1:  PR[GP1:91,1] = PR[GP1:90,1] + -19.923;
   1:  PR[GP1:91,2] = PR[GP1:90,2] + -17.300;
   1:L PR[91] 10mm/sec CNT100;
   1:  PR[GP1:91,1] = PR[GP1:90,1] + -19.075;
   1:  PR[GP1:91,2] = PR[GP1:90,2] + -17.702;
   1:L PR[91] 10mm/sec CNT100;
   1:  PR[GP1:91,1] = PR[GP1:90,1] + -16.522;
   1:  PR[GP1:91,2] = PR[GP1:90,2] + -18.860;
   1:L PR[91] 10mm/sec CNT100;
   1:  PR[GP1:91,1] = PR[GP1:90,1] + -13.902;
   1:  PR[GP1:91,2] = PR[GP1:90,2] + -19.699;
   1:L PR[91] 10mm/sec CNT100;
   1:  PR[GP1:91,1] = PR[GP1:90,1] + -13.520;
   1:  PR[GP1:91,2] = PR[GP1:90,2] + -19.805;
   1:L PR[91] 10mm/sec CNT100;
   1:  PR[GP1:91,1] = PR[GP1:90,1] + -12.954;
   1:  PR[GP1:91,2] = PR[GP1:90,2] + -19.909;
   1:L PR[91] 10mm/sec CNT100;
   1:  PR[GP1:91,1] = PR[GP1:90,1] + -10.056;
   1:  PR[GP1:91,2] = PR[GP1:90,2] + -20.529;
   1:L PR[91] 10mm/sec CNT100;
   1:  PR[GP1:91,1] = PR[GP1:90,1] + -7.500;
   1:  PR[GP1:91,2] = PR[GP1:90,2] + -20.755;
   1:L PR[91] 10mm/sec CNT100;
   1:  PR[GP1:91,1] = PR[GP1:90,1] + -5.731;
   1:  PR[GP1:91,2] = PR[GP1:90,2] + -20.848;
   1:L PR[91] 10mm/sec CNT100;
   1:  PR[GP1:91,1] = PR[GP1:90,1] + -3.765;
   1:  PR[GP1:91,2] = PR[GP1:90,2] + -20.776;
   1:L PR[91] 10mm/sec CNT100;
   1:  PR[GP1:91,1] = PR[GP1:90,1] + -0.700;
   1:  PR[GP1:91,2] = PR[GP1:90,2] + -20.337;
   1:L PR[91] 10mm/sec CNT100;
   1:  PR[GP1:91,1] = PR[GP1:90,1] + 0.482;
   1:  PR[GP1:91,2] = PR[GP1:90,2] + -20.129;
   1:L PR[91] 10mm/sec CNT100;
   1:  PR[GP1:91,1] = PR[GP1:90,1] + 1.704;
   1:  PR[GP1:91,2] = PR[GP1:90,2] + -19.711;
   1:L PR[91] 10mm/sec CNT100;
   1:  PR[GP1:91,1] = PR[GP1:90,1] + 2.072;
   1:  PR[GP1:91,2] = PR[GP1:90,2] + -19.622;
   1:L PR[91] 10mm/sec CNT100;
   1:  PR[GP1:91,1] = PR[GP1:90,1] + 3.416;
   1:  PR[GP1:91,2] = PR[GP1:90,2] + -19.796;
   1:L PR[91] 10mm/sec CNT100;
   1:  PR[GP1:91,1] = PR[GP1:90,1] + 5.423;
   1:  PR[GP1:91,2] = PR[GP1:90,2] + -20.487;
   1:L PR[91] 10mm/sec CNT100;
   1:  PR[GP1:91,1] = PR[GP1:90,1] + 5.646;
   1:  PR[GP1:91,2] = PR[GP1:90,2] + -20.559;
   1:L PR[91] 10mm/sec CNT100;
   1:  PR[GP1:91,1] = PR[GP1:90,1] + 6.118;
   1:  PR[GP1:91,2] = PR[GP1:90,2] + -20.669;
   1:L PR[91] 10mm/sec CNT100;
   1:  PR[GP1:91,1] = PR[GP1:90,1] + 8.398;
   1:  PR[GP1:91,2] = PR[GP1:90,2] + -21.069;
   1:L PR[91] 10mm/sec CNT100;
   1:  PR[GP1:91,1] = PR[GP1:90,1] + 8.759;
   1:  PR[GP1:91,2] = PR[GP1:90,2] + -21.092;
   1:L PR[91] 10mm/sec CNT100;
   1:  PR[GP1:91,1] = PR[GP1:90,1] + 11.208;
   1:  PR[GP1:91,2] = PR[GP1:90,2] + -21.116;
   1:L PR[91] 10mm/sec CNT100;
   1:  PR[GP1:91,1] = PR[GP1:90,1] + 14.042;
   1:  PR[GP1:91,2] = PR[GP1:90,2] + -20.696;
   1:L PR[91] 10mm/sec CNT100;
   1:  PR[GP1:91,1] = PR[GP1:90,1] + 16.799;
   1:  PR[GP1:91,2] = PR[GP1:90,2] + -19.833;
   1:L PR[91] 10mm/sec CNT100;
   1:  PR[GP1:91,1] = PR[GP1:90,1] + 19.410;
   1:  PR[GP1:91,2] = PR[GP1:90,2] + -18.534;
   1:L PR[91] 10mm/sec CNT100;
   1:  PR[GP1:91,1] = PR[GP1:90,1] + 21.804;
   1:  PR[GP1:91,2] = PR[GP1:90,2] + -16.826;
   1:L PR[91] 10mm/sec CNT100;
   1:  PR[GP1:91,1] = PR[GP1:90,1] + 23.522;
   1:  PR[GP1:91,2] = PR[GP1:90,2] + -15.141;
   1:L PR[91] 10mm/sec CNT100;
   1:  PR[GP1:91,1] = PR[GP1:90,1] + 23.972;
   1:  PR[GP1:91,2] = PR[GP1:90,2] + -14.717;
   1:L PR[91] 10mm/sec CNT100;
   1:  PR[GP1:91,1] = PR[GP1:90,1] + 25.384;
   1:  PR[GP1:91,2] = PR[GP1:90,2] + -12.963;
   1:L PR[91] 10mm/sec CNT100;
   1:  PR[GP1:91,1] = PR[GP1:90,1] + 25.887;
   1:  PR[GP1:91,2] = PR[GP1:90,2] + -12.268;
   1:L PR[91] 10mm/sec CNT100;
   1:  PR[GP1:91,1] = PR[GP1:90,1] + 26.608;
   1:  PR[GP1:91,2] = PR[GP1:90,2] + -11.029;
   1:L PR[91] 10mm/sec CNT100;
   1:  PR[GP1:91,1] = PR[GP1:90,1] + 27.329;
   1:  PR[GP1:91,2] = PR[GP1:90,2] + -9.662;
   1:L PR[91] 10mm/sec CNT100;
   1:  PR[GP1:91,1] = PR[GP1:90,1] + 27.583;
   1:  PR[GP1:91,2] = PR[GP1:90,2] + -9.019;
   1:L PR[91] 10mm/sec CNT100;
   1:  PR[GP1:91,1] = PR[GP1:90,1] + 28.306;
   1:  PR[GP1:91,2] = PR[GP1:90,2] + -7.005;
   1:L PR[91] 10mm/sec CNT100;
   1:  PR[GP1:91,1] = PR[GP1:90,1] + 28.875;
   1:  PR[GP1:91,2] = PR[GP1:90,2] + -4.413;
   1:L PR[91] 10mm/sec CNT100;
   1:  PR[GP1:91,1] = PR[GP1:90,1] + 29.013;
   1:  PR[GP1:91,2] = PR[GP1:90,2] + -1.809;
   1:L PR[91] 10mm/sec CNT100;
   1:  PR[GP1:91,1] = PR[GP1:90,1] + 28.593;
   1:  PR[GP1:91,2] = PR[GP1:90,2] + 1.620;
   1:L PR[91] 10mm/sec CNT100;
   1:  PR[GP1:91,1] = PR[GP1:90,1] + 27.492;
   1:  PR[GP1:91,2] = PR[GP1:90,2] + 4.844;
   1:L PR[91] 10mm/sec CNT100;
   1:  PR[GP1:91,1] = PR[GP1:90,1] + 25.750;
   1:  PR[GP1:91,2] = PR[GP1:90,2] + 7.749;
   1:L PR[91] 10mm/sec CNT100;
   1:  PR[GP1:91,1] = PR[GP1:90,1] + 23.442;
   1:  PR[GP1:91,2] = PR[GP1:90,2] + 10.236;
   1:L PR[91] 10mm/sec CNT100;
   1:  PR[GP1:91,1] = PR[GP1:90,1] + 22.362;
   1:  PR[GP1:91,2] = PR[GP1:90,2] + 11.008;
   1:L PR[91] 10mm/sec CNT100;
   1:  PR[GP1:91,1] = PR[GP1:90,1] + 20.660;
   1:  PR[GP1:91,2] = PR[GP1:90,2] + 12.219;
   1:L PR[91] 10mm/sec CNT100;
   1:  PR[GP1:91,1] = PR[GP1:90,1] + 17.495;
   1:  PR[GP1:91,2] = PR[GP1:90,2] + 13.636;
   1:L PR[91] 10mm/sec CNT100;
   1:  PR[GP1:91,1] = PR[GP1:90,1] + 14.134;
   1:  PR[GP1:91,2] = PR[GP1:90,2] + 14.415;
   1:L PR[91] 10mm/sec CNT100;
   1:  PR[GP1:91,1] = PR[GP1:90,1] + 10.649;
   1:  PR[GP1:91,2] = PR[GP1:90,2] + 14.552;
   1:L PR[91] 10mm/sec CNT100;
   1:  PR[GP1:91,1] = PR[GP1:90,1] + 9.158;
   1:  PR[GP1:91,2] = PR[GP1:90,2] + 14.338;
   1:L PR[91] 10mm/sec CNT100;
   1:  PR[GP1:91,1] = PR[GP1:90,1] + 7.206;
   1:  PR[GP1:91,2] = PR[GP1:90,2] + 14.034;
   1:L PR[91] 10mm/sec CNT100;
   1:  PR[GP1:91,1] = PR[GP1:90,1] + 3.868;
   1:  PR[GP1:91,2] = PR[GP1:90,2] + 12.889;
   1:L PR[91] 10mm/sec CNT100;
   1:  PR[GP1:91,1] = PR[GP1:90,1] + 1.906;
   1:  PR[GP1:91,2] = PR[GP1:90,2] + 11.864;
   1:L PR[91] 10mm/sec CNT100;
   1:  PR[GP1:91,1] = PR[GP1:90,1] + 1.359;
   1:  PR[GP1:91,2] = PR[GP1:90,2] + 11.722;
   1:L PR[91] 10mm/sec CNT100;
   1:  PR[GP1:91,1] = PR[GP1:90,1] + 0.620;
   1:  PR[GP1:91,2] = PR[GP1:90,2] + 11.498;
   1:L PR[91] 10mm/sec CNT100;
   1:  PR[GP1:91,1] = PR[GP1:90,1] + -0.423;
   1:  PR[GP1:91,2] = PR[GP1:90,2] + 11.731;
   1:L PR[91] 10mm/sec CNT100;
   1:  PR[GP1:91,1] = PR[GP1:90,1] + -1.504;
   1:  PR[GP1:91,2] = PR[GP1:90,2] + 12.174;
   1:L PR[91] 10mm/sec CNT100;
   1:  PR[GP1:91,1] = PR[GP1:90,1] + -4.240;
   1:  PR[GP1:91,2] = PR[GP1:90,2] + 13.112;
   1:L PR[91] 10mm/sec CNT100;
   1:  PR[GP1:91,1] = PR[GP1:90,1] + -7.352;
   1:  PR[GP1:91,2] = PR[GP1:90,2] + 13.835;
   1:L PR[91] 10mm/sec CNT100;
   1:  PR[GP1:91,1] = PR[GP1:90,1] + -8.796;
   1:  PR[GP1:91,2] = PR[GP1:90,2] + 14.003;
   1:L PR[91] 10mm/sec CNT100;
   1:  PR[GP1:91,1] = PR[GP1:90,1] + -11.350;
   1:  PR[GP1:91,2] = PR[GP1:90,2] + 14.214;
   1:L PR[91] 10mm/sec CNT100;
   1:  PR[GP1:91,1] = PR[GP1:90,1] + -11.845;
   1:  PR[GP1:91,2] = PR[GP1:90,2] + 14.217;
   1:L PR[91] 10mm/sec CNT100;
   1:  PR[GP1:91,1] = PR[GP1:90,1] + -15.242;
   1:  PR[GP1:91,2] = PR[GP1:90,2] + 13.951;
   1:L PR[91] 10mm/sec CNT100;
   1:  PR[GP1:91,1] = PR[GP1:90,1] + -15.947;
   1:  PR[GP1:91,2] = PR[GP1:90,2] + 13.817;
   1:L PR[91] 10mm/sec CNT100;
   1:  PR[GP1:91,1] = PR[GP1:90,1] + -18.471;
   1:  PR[GP1:91,2] = PR[GP1:90,2] + 13.152;
   1:L PR[91] 10mm/sec CNT100;
   1:  PR[GP1:91,1] = PR[GP1:90,1] + -20.213;
   1:  PR[GP1:91,2] = PR[GP1:90,2] + 12.455;
   1:L PR[91] 10mm/sec CNT100;
   1:  PR[GP1:91,1] = PR[GP1:90,1] + -21.606;
   1:  PR[GP1:91,2] = PR[GP1:90,2] + 11.792;
   1:L PR[91] 10mm/sec CNT100;
   1:  PR[GP1:91,1] = PR[GP1:90,1] + -23.857;
   1:  PR[GP1:91,2] = PR[GP1:90,2] + 10.304;
   1:L PR[91] 10mm/sec CNT100;
   1:  PR[GP1:91,1] = PR[GP1:90,1] + -24.465;
   1:  PR[GP1:91,2] = PR[GP1:90,2] + 9.847;
   1:L PR[91] 10mm/sec CNT100;
   1:  PR[GP1:91,1] = PR[GP1:90,1] + -26.681;
   1:  PR[GP1:91,2] = PR[GP1:90,2] + 7.542;
   1:L PR[91] 10mm/sec CNT100;
   1:  PR[GP1:91,1] = PR[GP1:90,1] + -26.854;
   1:  PR[GP1:91,2] = PR[GP1:90,2] + 7.341;
   1:L PR[91] 10mm/sec CNT100;
   1:  PR[GP1:91,1] = PR[GP1:90,1] + -28.639;
   1:  PR[GP1:91,2] = PR[GP1:90,2] + 4.343;
   1:L PR[91] 10mm/sec CNT100;
   1:  PR[GP1:91,1] = PR[GP1:90,1] + -29.720;
   1:  PR[GP1:91,2] = PR[GP1:90,2] + 1.047;
   1:L PR[91] 10mm/sec CNT100;
   1:  PR[GP1:91,1] = PR[GP1:90,1] + -29.899;
   1:  PR[GP1:91,2] = PR[GP1:90,2] + -2.320;
   1:L PR[91] 10mm/sec CNT100;
   1:  PR[GP1:91,1] = PR[GP1:90,1] + -29.917;
   1:  PR[GP1:91,2] = PR[GP1:90,2] + -2.485;
   1:L PR[91] 10mm/sec CNT100;
   1:  PR[GP1:91,1] = PR[GP1:90,1] + -29.485;
   1:  PR[GP1:91,2] = PR[GP1:90,2] + -4.950;
   1:L PR[91] 10mm/sec CNT100;
   1:  PR[GP1:91,1] = PR[GP1:90,1] + -29.346;
   1:  PR[GP1:91,2] = PR[GP1:90,2] + -5.525;
   1:L PR[91] 10mm/sec CNT100;
   1:  PR[GP1:91,1] = PR[GP1:90,1] + -29.245;
   1:  PR[GP1:91,2] = PR[GP1:90,2] + -6.057;
   1:L PR[91] 10mm/sec CNT100;
   1:  PR[GP1:91,1] = PR[GP1:90,1] + -27.880;
   1:  PR[GP1:91,2] = PR[GP1:90,2] + -9.438;
   1:L PR[91] 10mm/sec CNT100;
   1:  PR[GP1:91,1] = PR[GP1:90,1] + -26.990;
   1:  PR[GP1:91,2] = PR[GP1:90,2] + -10.764;
   1:L PR[91] 10mm/sec CNT100;
   1:  PR[GP1:91,1] = PR[GP1:90,1] + -25.782;
   1:  PR[GP1:91,2] = PR[GP1:90,2] + -12.503;
   1:L PR[91] 10mm/sec CNT100;
   1:  PR[GP1:91,1] = PR[GP1:90,1] + -23.731;
   1:  PR[GP1:91,2] = PR[GP1:90,2] + -14.558;
   1:L PR[91] 10mm/sec CNT100;
   1:  PR[GP1:91,1] = PR[GP1:90,1] + -22.578;
   1:  PR[GP1:91,2] = PR[GP1:90,2] + -15.244;
   1:  PR[GP1:91,3] = PR[GP1:90,3] + 34.100;
   1:L PR[91] 10mm/sec CNT100;
   1:  PR[GP1:91,1] = PR[GP1:90,1] + -19.155;
   1:  PR[GP1:91,2] = PR[GP1:90,2] + -17.509;
   1:L PR[91] 10mm/sec CNT100;
   1:  PR[GP1:91,1] = PR[GP1:90,1] + -17.209;
   1:  PR[GP1:91,2] = PR[GP1:90,2] + -18.430;
   1:L PR[91] 10mm/sec CNT100;
   1:  PR[GP1:91,1] = PR[GP1:90,1] + -15.931;
   1:  PR[GP1:91,2] = PR[GP1:90,2] + -19.010;
   1:L PR[91] 10mm/sec CNT100;
   1:  PR[GP1:91,1] = PR[GP1:90,1] + -14.102;
   1:  PR[GP1:91,2] = PR[GP1:90,2] + -19.596;
   1:L PR[91] 10mm/sec CNT100;
   1:  PR[GP1:91,1] = PR[GP1:90,1] + -12.868;
   1:  PR[GP1:91,2] = PR[GP1:90,2] + -20.024;
   1:L PR[91] 10mm/sec CNT100;
   1:  PR[GP1:91,1] = PR[GP1:90,1] + -12.424;
   1:  PR[GP1:91,2] = PR[GP1:90,2] + -20.130;
   1:L PR[91] 10mm/sec CNT100;
   1:  PR[GP1:91,1] = PR[GP1:90,1] + -9.136;
   1:  PR[GP1:91,2] = PR[GP1:90,2] + -20.834;
   1:L PR[91] 10mm/sec CNT100;
   1:  PR[GP1:91,1] = PR[GP1:90,1] + -6.947;
   1:  PR[GP1:91,2] = PR[GP1:90,2] + -21.027;
   1:L PR[91] 10mm/sec CNT100;
   1:  PR[GP1:91,1] = PR[GP1:90,1] + -4.569;
   1:  PR[GP1:91,2] = PR[GP1:90,2] + -21.152;
   1:L PR[91] 10mm/sec CNT100;
   1:  PR[GP1:91,1] = PR[GP1:90,1] + -3.036;
   1:  PR[GP1:91,2] = PR[GP1:90,2] + -21.096;
   1:L PR[91] 10mm/sec CNT100;
   1:  PR[GP1:91,1] = PR[GP1:90,1] + 0.716;
   1:  PR[GP1:91,2] = PR[GP1:90,2] + -20.559;
   1:L PR[91] 10mm/sec CNT100;
   1:  PR[GP1:91,1] = PR[GP1:90,1] + 1.414;
   1:  PR[GP1:91,2] = PR[GP1:90,2] + -20.436;
   1:L PR[91] 10mm/sec CNT100;
   1:  PR[GP1:91,1] = PR[GP1:90,1] + 2.369;
   1:  PR[GP1:91,2] = PR[GP1:90,2] + -20.126;
   1:L PR[91] 10mm/sec CNT100;
   1:  PR[GP1:91,1] = PR[GP1:90,1] + 3.741;
   1:  PR[GP1:91,2] = PR[GP1:90,2] + -20.267;
   1:L PR[91] 10mm/sec CNT100;
   1:  PR[GP1:91,1] = PR[GP1:90,1] + 5.357;
   1:  PR[GP1:91,2] = PR[GP1:90,2] + -20.801;
   1:L PR[91] 10mm/sec CNT100;
   1:  PR[GP1:91,1] = PR[GP1:90,1] + 6.538;
   1:  PR[GP1:91,2] = PR[GP1:90,2] + -21.076;
   1:L PR[91] 10mm/sec CNT100;
   1:  PR[GP1:91,1] = PR[GP1:90,1] + 8.094;
   1:  PR[GP1:91,2] = PR[GP1:90,2] + -21.349;
   1:L PR[91] 10mm/sec CNT100;
   1:  PR[GP1:91,1] = PR[GP1:90,1] + 9.241;
   1:  PR[GP1:91,2] = PR[GP1:90,2] + -21.422;
   1:L PR[91] 10mm/sec CNT100;
   1:  PR[GP1:91,1] = PR[GP1:90,1] + 10.911;
   1:  PR[GP1:91,2] = PR[GP1:90,2] + -21.438;
   1:L PR[91] 10mm/sec CNT100;
   1:  PR[GP1:91,1] = PR[GP1:90,1] + 11.901;
   1:  PR[GP1:91,2] = PR[GP1:90,2] + -21.336;
   1:L PR[91] 10mm/sec CNT100;
   1:  PR[GP1:91,1] = PR[GP1:90,1] + 13.744;
   1:  PR[GP1:91,2] = PR[GP1:90,2] + -21.050;
   1:L PR[91] 10mm/sec CNT100;
   1:  PR[GP1:91,1] = PR[GP1:90,1] + 14.439;
   1:  PR[GP1:91,2] = PR[GP1:90,2] + -20.860;
   1:L PR[91] 10mm/sec CNT100;
   1:  PR[GP1:91,1] = PR[GP1:90,1] + 16.515;
   1:  PR[GP1:91,2] = PR[GP1:90,2] + -20.178;
   1:L PR[91] 10mm/sec CNT100;
   1:  PR[GP1:91,1] = PR[GP1:90,1] + 16.795;
   1:  PR[GP1:91,2] = PR[GP1:90,2] + -20.050;
   1:L PR[91] 10mm/sec CNT100;
   1:  PR[GP1:91,1] = PR[GP1:90,1] + 18.256;
   1:  PR[GP1:91,2] = PR[GP1:90,2] + -19.292;
   1:L PR[91] 10mm/sec CNT100;
   1:  PR[GP1:91,1] = PR[GP1:90,1] + 19.137;
   1:  PR[GP1:91,2] = PR[GP1:90,2] + -18.858;
   1:L PR[91] 10mm/sec CNT100;
   1:  PR[GP1:91,1] = PR[GP1:90,1] + 21.539;
   1:  PR[GP1:91,2] = PR[GP1:90,2] + -17.167;
   1:L PR[91] 10mm/sec CNT100;
   1:  PR[GP1:91,1] = PR[GP1:90,1] + 23.658;
   1:  PR[GP1:91,2] = PR[GP1:90,2] + -15.112;
   1:L PR[91] 10mm/sec CNT100;
   1:  PR[GP1:91,1] = PR[GP1:90,1] + 25.436;
   1:  PR[GP1:91,2] = PR[GP1:90,2] + -12.741;
   1:L PR[91] 10mm/sec CNT100;
   1:  PR[GP1:91,1] = PR[GP1:90,1] + 26.656;
   1:  PR[GP1:91,2] = PR[GP1:90,2] + -10.622;
   1:L PR[91] 10mm/sec CNT100;
   1:  PR[GP1:91,1] = PR[GP1:90,1] + 26.932;
   1:  PR[GP1:91,2] = PR[GP1:90,2] + -10.101;
   1:L PR[91] 10mm/sec CNT100;
   1:  PR[GP1:91,1] = PR[GP1:90,1] + 27.558;
   1:  PR[GP1:91,2] = PR[GP1:90,2] + -8.518;
   1:L PR[91] 10mm/sec CNT100;
   1:  PR[GP1:91,1] = PR[GP1:90,1] + 27.965;
   1:  PR[GP1:91,2] = PR[GP1:90,2] + -7.384;
   1:L PR[91] 10mm/sec CNT100;
   1:  PR[GP1:91,1] = PR[GP1:90,1] + 28.197;
   1:  PR[GP1:91,2] = PR[GP1:90,2] + -6.361;
   1:L PR[91] 10mm/sec CNT100;
   1:  PR[GP1:91,1] = PR[GP1:90,1] + 28.536;
   1:  PR[GP1:91,2] = PR[GP1:90,2] + -4.679;
   1:L PR[91] 10mm/sec CNT100;
   1:  PR[GP1:91,1] = PR[GP1:90,1] + 28.657;
   1:  PR[GP1:91,2] = PR[GP1:90,2] + -2.014;
   1:L PR[91] 10mm/sec CNT100;
   1:  PR[GP1:91,1] = PR[GP1:90,1] + 28.248;
   1:  PR[GP1:91,2] = PR[GP1:90,2] + 1.422;
   1:L PR[91] 10mm/sec CNT100;
   1:  PR[GP1:91,1] = PR[GP1:90,1] + 27.152;
   1:  PR[GP1:91,2] = PR[GP1:90,2] + 4.652;
   1:L PR[91] 10mm/sec CNT100;
   1:  PR[GP1:91,1] = PR[GP1:90,1] + 25.408;
   1:  PR[GP1:91,2] = PR[GP1:90,2] + 7.566;
   1:L PR[91] 10mm/sec CNT100;
   1:  PR[GP1:91,1] = PR[GP1:90,1] + 23.095;
   1:  PR[GP1:91,2] = PR[GP1:90,2] + 10.062;
   1:L PR[91] 10mm/sec CNT100;
   1:  PR[GP1:91,1] = PR[GP1:90,1] + 20.305;
   1:  PR[GP1:91,2] = PR[GP1:90,2] + 12.054;
   1:L PR[91] 10mm/sec CNT100;
   1:  PR[GP1:91,1] = PR[GP1:90,1] + 17.172;
   1:  PR[GP1:91,2] = PR[GP1:90,2] + 13.463;
   1:L PR[91] 10mm/sec CNT100;
   1:  PR[GP1:91,1] = PR[GP1:90,1] + 13.848;
   1:  PR[GP1:91,2] = PR[GP1:90,2] + 14.236;
   1:L PR[91] 10mm/sec CNT100;
   1:  PR[GP1:91,1] = PR[GP1:90,1] + 10.402;
   1:  PR[GP1:91,2] = PR[GP1:90,2] + 14.368;
   1:L PR[91] 10mm/sec CNT100;
   1:  PR[GP1:91,1] = PR[GP1:90,1] + 6.910;
   1:  PR[GP1:91,2] = PR[GP1:90,2] + 13.869;
   1:L PR[91] 10mm/sec CNT100;
   1:  PR[GP1:91,1] = PR[GP1:90,1] + 3.533;
   1:  PR[GP1:91,2] = PR[GP1:90,2] + 12.662;
   1:L PR[91] 10mm/sec CNT100;
   1:  PR[GP1:91,1] = PR[GP1:90,1] + 3.037;
   1:  PR[GP1:91,2] = PR[GP1:90,2] + 12.423;
   1:L PR[91] 10mm/sec CNT100;
   1:  PR[GP1:91,1] = PR[GP1:90,1] + 2.080;
   1:  PR[GP1:91,2] = PR[GP1:90,2] + 11.928;
   1:L PR[91] 10mm/sec CNT100;
   1:  PR[GP1:91,1] = PR[GP1:90,1] + 0.774;
   1:  PR[GP1:91,2] = PR[GP1:90,2] + 11.599;
   1:L PR[91] 10mm/sec CNT100;
   1:  PR[GP1:91,1] = PR[GP1:90,1] + -0.163;
   1:  PR[GP1:91,2] = PR[GP1:90,2] + 11.802;
   1:L PR[91] 10mm/sec CNT100;
   1:  PR[GP1:91,1] = PR[GP1:90,1] + -0.724;
   1:  PR[GP1:91,2] = PR[GP1:90,2] + 12.019;
   1:L PR[91] 10mm/sec CNT100;
   1:  PR[GP1:91,1] = PR[GP1:90,1] + -3.034;
   1:  PR[GP1:91,2] = PR[GP1:90,2] + 12.805;
   1:L PR[91] 10mm/sec CNT100;
   1:  PR[GP1:91,1] = PR[GP1:90,1] + -3.318;
   1:  PR[GP1:91,2] = PR[GP1:90,2] + 12.890;
   1:L PR[91] 10mm/sec CNT100;
   1:  PR[GP1:91,1] = PR[GP1:90,1] + -6.503;
   1:  PR[GP1:91,2] = PR[GP1:90,2] + 13.641;
   1:L PR[91] 10mm/sec CNT100;
   1:  PR[GP1:91,1] = PR[GP1:90,1] + -8.549;
   1:  PR[GP1:91,2] = PR[GP1:90,2] + 13.879;
   1:L PR[91] 10mm/sec CNT100;
   1:  PR[GP1:91,1] = PR[GP1:90,1] + -10.162;
   1:  PR[GP1:91,2] = PR[GP1:90,2] + 14.013;
   1:L PR[91] 10mm/sec CNT100;
   1:  PR[GP1:91,1] = PR[GP1:90,1] + -11.392;
   1:  PR[GP1:91,2] = PR[GP1:90,2] + 14.020;
   1:L PR[91] 10mm/sec CNT100;
   1:  PR[GP1:91,1] = PR[GP1:90,1] + -14.885;
   1:  PR[GP1:91,2] = PR[GP1:90,2] + 13.746;
   1:L PR[91] 10mm/sec CNT100;
   1:  PR[GP1:91,1] = PR[GP1:90,1] + -18.118;
   1:  PR[GP1:91,2] = PR[GP1:90,2] + 12.900;
   1:L PR[91] 10mm/sec CNT100;
   1:  PR[GP1:91,1] = PR[GP1:90,1] + -19.091;
   1:  PR[GP1:91,2] = PR[GP1:90,2] + 12.511;
   1:L PR[91] 10mm/sec CNT100;
   1:  PR[GP1:91,1] = PR[GP1:90,1] + -21.186;
   1:  PR[GP1:91,2] = PR[GP1:90,2] + 11.513;
   1:L PR[91] 10mm/sec CNT100;
   1:  PR[GP1:91,1] = PR[GP1:90,1] + -22.793;
   1:  PR[GP1:91,2] = PR[GP1:90,2] + 10.450;
   1:L PR[91] 10mm/sec CNT100;
   1:  PR[GP1:91,1] = PR[GP1:90,1] + -23.982;
   1:  PR[GP1:91,2] = PR[GP1:90,2] + 9.559;
   1:L PR[91] 10mm/sec CNT100;
   1:  PR[GP1:91,1] = PR[GP1:90,1] + -25.702;
   1:  PR[GP1:91,2] = PR[GP1:90,2] + 7.769;
   1:L PR[91] 10mm/sec CNT100;
   1:  PR[GP1:91,1] = PR[GP1:90,1] + -26.316;
   1:  PR[GP1:91,2] = PR[GP1:90,2] + 7.057;
   1:L PR[91] 10mm/sec CNT100;
   1:  PR[GP1:91,1] = PR[GP1:90,1] + -27.739;
   1:  PR[GP1:91,2] = PR[GP1:90,2] + 4.673;
   1:L PR[91] 10mm/sec CNT100;
   1:  PR[GP1:91,1] = PR[GP1:90,1] + -28.055;
   1:  PR[GP1:91,2] = PR[GP1:90,2] + 4.091;
   1:L PR[91] 10mm/sec CNT100;
   1:  PR[GP1:91,1] = PR[GP1:90,1] + -28.947;
   1:  PR[GP1:91,2] = PR[GP1:90,2] + 1.375;
   1:L PR[91] 10mm/sec CNT100;
   1:  PR[GP1:91,1] = PR[GP1:90,1] + -29.113;
   1:  PR[GP1:91,2] = PR[GP1:90,2] + 0.821;
   1:L PR[91] 10mm/sec CNT100;
   1:  PR[GP1:91,1] = PR[GP1:90,1] + -29.259;
   1:  PR[GP1:91,2] = PR[GP1:90,2] + -1.946;
   1:L PR[91] 10mm/sec CNT100;
   1:  PR[GP1:91,1] = PR[GP1:90,1] + -29.339;
   1:  PR[GP1:91,2] = PR[GP1:90,2] + -2.675;
   1:L PR[91] 10mm/sec CNT100;
   1:  PR[GP1:91,1] = PR[GP1:90,1] + -29.109;
   1:  PR[GP1:91,2] = PR[GP1:90,2] + -3.986;
   1:L PR[91] 10mm/sec CNT100;
   1:  PR[GP1:91,1] = PR[GP1:90,1] + -28.834;
   1:  PR[GP1:91,2] = PR[GP1:90,2] + -5.129;
   1:L PR[91] 10mm/sec CNT100;
   1:  PR[GP1:91,1] = PR[GP1:90,1] + -28.625;
   1:  PR[GP1:91,2] = PR[GP1:90,2] + -6.229;
   1:L PR[91] 10mm/sec CNT100;
   1:  PR[GP1:91,1] = PR[GP1:90,1] + -27.280;
   1:  PR[GP1:91,2] = PR[GP1:90,2] + -9.579;
   1:L PR[91] 10mm/sec CNT100;
   1:  PR[GP1:91,1] = PR[GP1:90,1] + -25.898;
   1:  PR[GP1:91,2] = PR[GP1:90,2] + -11.638;
   1:L PR[91] 10mm/sec CNT100;
   1:  PR[GP1:91,1] = PR[GP1:90,1] + -25.218;
   1:  PR[GP1:91,2] = PR[GP1:90,2] + -12.617;
   1:L PR[91] 10mm/sec CNT100;
   1:  PR[GP1:91,1] = PR[GP1:90,1] + -22.850;
   1:  PR[GP1:91,2] = PR[GP1:90,2] + -14.991;
   1:L PR[91] 10mm/sec CNT100;
   1:  PR[GP1:91,1] = PR[GP1:90,1] + -21.670;
   1:  PR[GP1:91,2] = PR[GP1:90,2] + -15.554;
   1:  PR[GP1:91,3] = PR[GP1:90,3] + 35.200;
   1:L PR[91] 10mm/sec CNT100;
   1:  PR[GP1:91,1] = PR[GP1:90,1] + -19.683;
   1:  PR[GP1:91,2] = PR[GP1:90,2] + -16.876;
   1:L PR[91] 10mm/sec CNT100;
   1:  PR[GP1:91,1] = PR[GP1:90,1] + -18.390;
   1:  PR[GP1:91,2] = PR[GP1:90,2] + -17.716;
   1:L PR[91] 10mm/sec CNT100;
   1:  PR[GP1:91,1] = PR[GP1:90,1] + -15.328;
   1:  PR[GP1:91,2] = PR[GP1:90,2] + -19.164;
   1:L PR[91] 10mm/sec CNT100;
   1:  PR[GP1:91,1] = PR[GP1:90,1] + -12.145;
   1:  PR[GP1:91,2] = PR[GP1:90,2] + -20.268;
   1:L PR[91] 10mm/sec CNT100;
   1:  PR[GP1:91,1] = PR[GP1:90,1] + -10.959;
   1:  PR[GP1:91,2] = PR[GP1:90,2] + -20.552;
   1:L PR[91] 10mm/sec CNT100;
   1:  PR[GP1:91,1] = PR[GP1:90,1] + -8.216;
   1:  PR[GP1:91,2] = PR[GP1:90,2] + -21.139;
   1:L PR[91] 10mm/sec CNT100;
   1:  PR[GP1:91,1] = PR[GP1:90,1] + -6.393;
   1:  PR[GP1:91,2] = PR[GP1:90,2] + -21.300;
   1:L PR[91] 10mm/sec CNT100;
   1:  PR[GP1:91,1] = PR[GP1:90,1] + -3.407;
   1:  PR[GP1:91,2] = PR[GP1:90,2] + -21.457;
   1:L PR[91] 10mm/sec CNT100;
   1:  PR[GP1:91,1] = PR[GP1:90,1] + -2.307;
   1:  PR[GP1:91,2] = PR[GP1:90,2] + -21.417;
   1:L PR[91] 10mm/sec CNT100;
   1:  PR[GP1:91,1] = PR[GP1:90,1] + 2.132;
   1:  PR[GP1:91,2] = PR[GP1:90,2] + -20.781;
   1:L PR[91] 10mm/sec CNT100;
   1:  PR[GP1:91,1] = PR[GP1:90,1] + 2.340;
   1:  PR[GP1:91,2] = PR[GP1:90,2] + -20.744;
   1:L PR[91] 10mm/sec CNT100;
   1:  PR[GP1:91,1] = PR[GP1:90,1] + 2.712;
   1:  PR[GP1:91,2] = PR[GP1:90,2] + -20.623;
   1:L PR[91] 10mm/sec CNT100;
   1:  PR[GP1:91,1] = PR[GP1:90,1] + 4.087;
   1:  PR[GP1:91,2] = PR[GP1:90,2] + -20.729;
   1:L PR[91] 10mm/sec CNT100;
   1:  PR[GP1:91,1] = PR[GP1:90,1] + 5.063;
   1:  PR[GP1:91,2] = PR[GP1:90,2] + -21.042;
   1:L PR[91] 10mm/sec CNT100;
   1:  PR[GP1:91,1] = PR[GP1:90,1] + 6.958;
   1:  PR[GP1:91,2] = PR[GP1:90,2] + -21.483;
   1:L PR[91] 10mm/sec CNT100;
   1:  PR[GP1:91,1] = PR[GP1:90,1] + 7.791;
   1:  PR[GP1:91,2] = PR[GP1:90,2] + -21.629;
   1:L PR[91] 10mm/sec CNT100;
   1:  PR[GP1:91,1] = PR[GP1:90,1] + 9.723;
   1:  PR[GP1:91,2] = PR[GP1:90,2] + -21.751;
   1:L PR[91] 10mm/sec CNT100;
   1:  PR[GP1:91,1] = PR[GP1:90,1] + 10.600;
   1:  PR[GP1:91,2] = PR[GP1:90,2] + -21.759;
   1:L PR[91] 10mm/sec CNT100;
   1:  PR[GP1:91,1] = PR[GP1:90,1] + 12.438;
   1:  PR[GP1:91,2] = PR[GP1:90,2] + -21.571;
   1:L PR[91] 10mm/sec CNT100;
   1:  PR[GP1:91,1] = PR[GP1:90,1] + 13.431;
   1:  PR[GP1:91,2] = PR[GP1:90,2] + -21.416;
   1:L PR[91] 10mm/sec CNT100;
   1:  PR[GP1:91,1] = PR[GP1:90,1] + 15.018;
   1:  PR[GP1:91,2] = PR[GP1:90,2] + -20.982;
   1:L PR[91] 10mm/sec CNT100;
   1:  PR[GP1:91,1] = PR[GP1:90,1] + 16.209;
   1:  PR[GP1:91,2] = PR[GP1:90,2] + -20.591;
   1:L PR[91] 10mm/sec CNT100;
   1:  PR[GP1:91,1] = PR[GP1:90,1] + 17.399;
   1:  PR[GP1:91,2] = PR[GP1:90,2] + -20.046;
   1:L PR[91] 10mm/sec CNT100;
   1:  PR[GP1:91,1] = PR[GP1:90,1] + 18.852;
   1:  PR[GP1:91,2] = PR[GP1:90,2] + -19.292;
   1:L PR[91] 10mm/sec CNT100;
   1:  PR[GP1:91,1] = PR[GP1:90,1] + 19.535;
   1:  PR[GP1:91,2] = PR[GP1:90,2] + -18.833;
   1:L PR[91] 10mm/sec CNT100;
   1:  PR[GP1:91,1] = PR[GP1:90,1] + 21.263;
   1:  PR[GP1:91,2] = PR[GP1:90,2] + -17.552;
   1:L PR[91] 10mm/sec CNT100;
   1:  PR[GP1:91,1] = PR[GP1:90,1] + 21.963;
   1:  PR[GP1:91,2] = PR[GP1:90,2] + -16.853;
   1:L PR[91] 10mm/sec CNT100;
   1:  PR[GP1:91,1] = PR[GP1:90,1] + 23.405;
   1:  PR[GP1:91,2] = PR[GP1:90,2] + -15.469;
   1:L PR[91] 10mm/sec CNT100;
   1:  PR[GP1:91,1] = PR[GP1:90,1] + 25.191;
   1:  PR[GP1:91,2] = PR[GP1:90,2] + -13.120;
   1:L PR[91] 10mm/sec CNT100;
   1:  PR[GP1:91,1] = PR[GP1:90,1] + 26.589;
   1:  PR[GP1:91,2] = PR[GP1:90,2] + -10.528;
   1:L PR[91] 10mm/sec CNT100;
   1:  PR[GP1:91,1] = PR[GP1:90,1] + 27.084;
   1:  PR[GP1:91,2] = PR[GP1:90,2] + -9.152;
   1:L PR[91] 10mm/sec CNT100;
   1:  PR[GP1:91,1] = PR[GP1:90,1] + 27.532;
   1:  PR[GP1:91,2] = PR[GP1:90,2] + -8.017;
   1:L PR[91] 10mm/sec CNT100;
   1:  PR[GP1:91,1] = PR[GP1:90,1] + 27.623;
   1:  PR[GP1:91,2] = PR[GP1:90,2] + -7.766;
   1:L PR[91] 10mm/sec CNT100;
   1:  PR[GP1:91,1] = PR[GP1:90,1] + 28.073;
   1:  PR[GP1:91,2] = PR[GP1:90,2] + -5.780;
   1:L PR[91] 10mm/sec CNT100;
   1:  PR[GP1:91,1] = PR[GP1:90,1] + 28.230;
   1:  PR[GP1:91,2] = PR[GP1:90,2] + -5.000;
   1:L PR[91] 10mm/sec CNT100;
   1:  PR[GP1:91,1] = PR[GP1:90,1] + 28.341;
   1:  PR[GP1:91,2] = PR[GP1:90,2] + -2.253;
   1:L PR[91] 10mm/sec CNT100;
   1:  PR[GP1:91,1] = PR[GP1:90,1] + 27.904;
   1:  PR[GP1:91,2] = PR[GP1:90,2] + 1.221;
   1:L PR[91] 10mm/sec CNT100;
   1:  PR[GP1:91,1] = PR[GP1:90,1] + 26.812;
   1:  PR[GP1:91,2] = PR[GP1:90,2] + 4.461;
   1:L PR[91] 10mm/sec CNT100;
   1:  PR[GP1:91,1] = PR[GP1:90,1] + 25.066;
   1:  PR[GP1:91,2] = PR[GP1:90,2] + 7.383;
   1:L PR[91] 10mm/sec CNT100;
   1:  PR[GP1:91,1] = PR[GP1:90,1] + 22.747;
   1:  PR[GP1:91,2] = PR[GP1:90,2] + 9.889;
   1:L PR[91] 10mm/sec CNT100;
   1:  PR[GP1:91,1] = PR[GP1:90,1] + 19.995;
   1:  PR[GP1:91,2] = PR[GP1:90,2] + 11.871;
   1:L PR[91] 10mm/sec CNT100;
   1:  PR[GP1:91,1] = PR[GP1:90,1] + 16.917;
   1:  PR[GP1:91,2] = PR[GP1:90,2] + 13.267;
   1:L PR[91] 10mm/sec CNT100;
   1:  PR[GP1:91,1] = PR[GP1:90,1] + 13.561;
   1:  PR[GP1:91,2] = PR[GP1:90,2] + 14.057;
   1:L PR[91] 10mm/sec CNT100;
   1:  PR[GP1:91,1] = PR[GP1:90,1] + 10.154;
   1:  PR[GP1:91,2] = PR[GP1:90,2] + 14.185;
   1:L PR[91] 10mm/sec CNT100;
   1:  PR[GP1:91,1] = PR[GP1:90,1] + 8.027;
   1:  PR[GP1:91,2] = PR[GP1:90,2] + 13.881;
   1:L PR[91] 10mm/sec CNT100;
   1:  PR[GP1:91,1] = PR[GP1:90,1] + 6.742;
   1:  PR[GP1:91,2] = PR[GP1:90,2] + 13.677;
   1:L PR[91] 10mm/sec CNT100;
   1:  PR[GP1:91,1] = PR[GP1:90,1] + 3.461;
   1:  PR[GP1:91,2] = PR[GP1:90,2] + 12.517;
   1:L PR[91] 10mm/sec CNT100;
   1:  PR[GP1:91,1] = PR[GP1:90,1] + 3.205;
   1:  PR[GP1:91,2] = PR[GP1:90,2] + 12.416;
   1:L PR[91] 10mm/sec CNT100;
   1:  PR[GP1:91,1] = PR[GP1:90,1] + 2.243;
   1:  PR[GP1:91,2] = PR[GP1:90,2] + 11.954;
   1:L PR[91] 10mm/sec CNT100;
   1:  PR[GP1:91,1] = PR[GP1:90,1] + 1.887;
   1:  PR[GP1:91,2] = PR[GP1:90,2] + 11.883;
   1:L PR[91] 10mm/sec CNT100;
   1:  PR[GP1:91,1] = PR[GP1:90,1] + 0.952;
   1:  PR[GP1:91,2] = PR[GP1:90,2] + 11.652;
   1:L PR[91] 10mm/sec CNT100;
   1:  PR[GP1:91,1] = PR[GP1:90,1] + 0.109;
   1:  PR[GP1:91,2] = PR[GP1:90,2] + 11.845;
   1:L PR[91] 10mm/sec CNT100;
   1:  PR[GP1:91,1] = PR[GP1:90,1] + -1.808;
   1:  PR[GP1:91,2] = PR[GP1:90,2] + 12.492;
   1:L PR[91] 10mm/sec CNT100;
   1:  PR[GP1:91,1] = PR[GP1:90,1] + -2.356;
   1:  PR[GP1:91,2] = PR[GP1:90,2] + 12.656;
   1:L PR[91] 10mm/sec CNT100;
   1:  PR[GP1:91,1] = PR[GP1:90,1] + -5.431;
   1:  PR[GP1:91,2] = PR[GP1:90,2] + 13.385;
   1:L PR[91] 10mm/sec CNT100;
   1:  PR[GP1:91,1] = PR[GP1:90,1] + -5.819;
   1:  PR[GP1:91,2] = PR[GP1:90,2] + 13.451;
   1:L PR[91] 10mm/sec CNT100;
   1:  PR[GP1:91,1] = PR[GP1:90,1] + -7.157;
   1:  PR[GP1:91,2] = PR[GP1:90,2] + 13.622;
   1:L PR[91] 10mm/sec CNT100;
   1:  PR[GP1:91,1] = PR[GP1:90,1] + -8.303;
   1:  PR[GP1:91,2] = PR[GP1:90,2] + 13.755;
   1:L PR[91] 10mm/sec CNT100;
   1:  PR[GP1:91,1] = PR[GP1:90,1] + -8.974;
   1:  PR[GP1:91,2] = PR[GP1:90,2] + 13.811;
   1:L PR[91] 10mm/sec CNT100;
   1:  PR[GP1:91,1] = PR[GP1:90,1] + -10.940;
   1:  PR[GP1:91,2] = PR[GP1:90,2] + 13.823;
   1:L PR[91] 10mm/sec CNT100;
   1:  PR[GP1:91,1] = PR[GP1:90,1] + -13.280;
   1:  PR[GP1:91,2] = PR[GP1:90,2] + 13.642;
   1:L PR[91] 10mm/sec CNT100;
   1:  PR[GP1:91,1] = PR[GP1:90,1] + -14.193;
   1:  PR[GP1:91,2] = PR[GP1:90,2] + 13.538;
   1:L PR[91] 10mm/sec CNT100;
   1:  PR[GP1:91,1] = PR[GP1:90,1] + -17.048;
   1:  PR[GP1:91,2] = PR[GP1:90,2] + 12.837;
   1:L PR[91] 10mm/sec CNT100;
   1:  PR[GP1:91,1] = PR[GP1:90,1] + -17.765;
   1:  PR[GP1:91,2] = PR[GP1:90,2] + 12.648;
   1:L PR[91] 10mm/sec CNT100;
   1:  PR[GP1:91,1] = PR[GP1:90,1] + -17.969;
   1:  PR[GP1:91,2] = PR[GP1:90,2] + 12.566;
   1:L PR[91] 10mm/sec CNT100;
   1:  PR[GP1:91,1] = PR[GP1:90,1] + -20.766;
   1:  PR[GP1:91,2] = PR[GP1:90,2] + 11.234;
   1:L PR[91] 10mm/sec CNT100;
   1:  PR[GP1:91,1] = PR[GP1:90,1] + -21.731;
   1:  PR[GP1:91,2] = PR[GP1:90,2] + 10.596;
   1:L PR[91] 10mm/sec CNT100;
   1:  PR[GP1:91,1] = PR[GP1:90,1] + -23.499;
   1:  PR[GP1:91,2] = PR[GP1:90,2] + 9.270;
   1:L PR[91] 10mm/sec CNT100;
   1:  PR[GP1:91,1] = PR[GP1:90,1] + -24.723;
   1:  PR[GP1:91,2] = PR[GP1:90,2] + 7.996;
   1:L PR[91] 10mm/sec CNT100;
   1:  PR[GP1:91,1] = PR[GP1:90,1] + -25.778;
   1:  PR[GP1:91,2] = PR[GP1:90,2] + 6.773;
   1:L PR[91] 10mm/sec CNT100;
   1:  PR[GP1:91,1] = PR[GP1:90,1] + -26.856;
   1:  PR[GP1:91,2] = PR[GP1:90,2] + 4.966;
   1:L PR[91] 10mm/sec CNT100;
   1:  PR[GP1:91,1] = PR[GP1:90,1] + -27.475;
   1:  PR[GP1:91,2] = PR[GP1:90,2] + 3.826;
   1:L PR[91] 10mm/sec CNT100;
   1:  PR[GP1:91,1] = PR[GP1:90,1] + -28.168;
   1:  PR[GP1:91,2] = PR[GP1:90,2] + 1.715;
   1:L PR[91] 10mm/sec CNT100;
   1:  PR[GP1:91,1] = PR[GP1:90,1] + -28.506;
   1:  PR[GP1:91,2] = PR[GP1:90,2] + 0.585;
   1:L PR[91] 10mm/sec CNT100;
   1:  PR[GP1:91,1] = PR[GP1:90,1] + -28.620;
   1:  PR[GP1:91,2] = PR[GP1:90,2] + -1.572;
   1:L PR[91] 10mm/sec CNT100;
   1:  PR[GP1:91,1] = PR[GP1:90,1] + -28.762;
   1:  PR[GP1:91,2] = PR[GP1:90,2] + -2.864;
   1:L PR[91] 10mm/sec CNT100;
   1:  PR[GP1:91,1] = PR[GP1:90,1] + -28.734;
   1:  PR[GP1:91,2] = PR[GP1:90,2] + -3.023;
   1:L PR[91] 10mm/sec CNT100;
   1:  PR[GP1:91,1] = PR[GP1:90,1] + -28.322;
   1:  PR[GP1:91,2] = PR[GP1:90,2] + -4.734;
   1:L PR[91] 10mm/sec CNT100;
   1:  PR[GP1:91,1] = PR[GP1:90,1] + -28.004;
   1:  PR[GP1:91,2] = PR[GP1:90,2] + -6.401;
   1:L PR[91] 10mm/sec CNT100;
   1:  PR[GP1:91,1] = PR[GP1:90,1] + -26.681;
   1:  PR[GP1:91,2] = PR[GP1:90,2] + -9.719;
   1:L PR[91] 10mm/sec CNT100;
   1:  PR[GP1:91,1] = PR[GP1:90,1] + -24.651;
   1:  PR[GP1:91,2] = PR[GP1:90,2] + -12.734;
   1:L PR[91] 10mm/sec CNT100;
   1:  PR[GP1:91,1] = PR[GP1:90,1] + -24.069;
   1:  PR[GP1:91,2] = PR[GP1:90,2] + -13.318;
   1:L PR[91] 10mm/sec CNT100;
   1:  PR[GP1:91,1] = PR[GP1:90,1] + -22.171;
   1:  PR[GP1:91,2] = PR[GP1:90,2] + -15.125;
   1:L PR[91] 10mm/sec CNT100;
   1:  PR[GP1:91,1] = PR[GP1:90,1] + -20.751;
   1:  PR[GP1:91,2] = PR[GP1:90,2] + -15.870;
   1:  PR[GP1:91,3] = PR[GP1:90,3] + 36.300;
   1:L PR[91] 10mm/sec CNT100;
   1:  PR[GP1:91,1] = PR[GP1:90,1] + -19.389;
   1:  PR[GP1:91,2] = PR[GP1:90,2] + -16.777;
   1:L PR[91] 10mm/sec CNT100;
   1:  PR[GP1:91,1] = PR[GP1:90,1] + -17.621;
   1:  PR[GP1:91,2] = PR[GP1:90,2] + -17.926;
   1:L PR[91] 10mm/sec CNT100;
   1:  PR[GP1:91,1] = PR[GP1:90,1] + -14.719;
   1:  PR[GP1:91,2] = PR[GP1:90,2] + -19.321;
   1:L PR[91] 10mm/sec CNT100;
   1:  PR[GP1:91,1] = PR[GP1:90,1] + -14.207;
   1:  PR[GP1:91,2] = PR[GP1:90,2] + -19.545;
   1:L PR[91] 10mm/sec CNT100;
   1:  PR[GP1:91,1] = PR[GP1:90,1] + -11.422;
   1:  PR[GP1:91,2] = PR[GP1:90,2] + -20.513;
   1:L PR[91] 10mm/sec CNT100;
   1:  PR[GP1:91,1] = PR[GP1:90,1] + -9.494;
   1:  PR[GP1:91,2] = PR[GP1:90,2] + -20.974;
   1:L PR[91] 10mm/sec CNT100;
   1:  PR[GP1:91,1] = PR[GP1:90,1] + -7.296;
   1:  PR[GP1:91,2] = PR[GP1:90,2] + -21.444;
   1:L PR[91] 10mm/sec CNT100;
   1:  PR[GP1:91,1] = PR[GP1:90,1] + -5.840;
   1:  PR[GP1:91,2] = PR[GP1:90,2] + -21.573;
   1:L PR[91] 10mm/sec CNT100;
   1:  PR[GP1:91,1] = PR[GP1:90,1] + -2.245;
   1:  PR[GP1:91,2] = PR[GP1:90,2] + -21.761;
   1:L PR[91] 10mm/sec CNT100;
   1:  PR[GP1:91,1] = PR[GP1:90,1] + -1.578;
   1:  PR[GP1:91,2] = PR[GP1:90,2] + -21.737;
   1:L PR[91] 10mm/sec CNT100;
   1:  PR[GP1:91,1] = PR[GP1:90,1] + 2.224;
   1:  PR[GP1:91,2] = PR[GP1:90,2] + -21.193;
   1:L PR[91] 10mm/sec CNT100;
   1:  PR[GP1:91,1] = PR[GP1:90,1] + 3.208;
   1:  PR[GP1:91,2] = PR[GP1:90,2] + -21.104;
   1:L PR[91] 10mm/sec CNT100;
   1:  PR[GP1:91,1] = PR[GP1:90,1] + 4.458;
   1:  PR[GP1:91,2] = PR[GP1:90,2] + -21.185;
   1:L PR[91] 10mm/sec CNT100;
   1:  PR[GP1:91,1] = PR[GP1:90,1] + 4.768;
   1:  PR[GP1:91,2] = PR[GP1:90,2] + -21.283;
   1:L PR[91] 10mm/sec CNT100;
   1:  PR[GP1:91,1] = PR[GP1:90,1] + 7.503;
   1:  PR[GP1:91,2] = PR[GP1:90,2] + -21.910;
   1:L PR[91] 10mm/sec CNT100;
   1:  PR[GP1:91,1] = PR[GP1:90,1] + 10.304;
   1:  PR[GP1:91,2] = PR[GP1:90,2] + -22.080;
   1:L PR[91] 10mm/sec CNT100;
   1:  PR[GP1:91,1] = PR[GP1:90,1] + 13.134;
   1:  PR[GP1:91,2] = PR[GP1:90,2] + -21.779;
   1:L PR[91] 10mm/sec CNT100;
   1:  PR[GP1:91,1] = PR[GP1:90,1] + 15.598;
   1:  PR[GP1:91,2] = PR[GP1:90,2] + -21.105;
   1:L PR[91] 10mm/sec CNT100;
   1:  PR[GP1:91,1] = PR[GP1:90,1] + 15.904;
   1:  PR[GP1:91,2] = PR[GP1:90,2] + -21.004;
   1:L PR[91] 10mm/sec CNT100;
   1:  PR[GP1:91,1] = PR[GP1:90,1] + 18.003;
   1:  PR[GP1:91,2] = PR[GP1:90,2] + -20.042;
   1:L PR[91] 10mm/sec CNT100;
   1:  PR[GP1:91,1] = PR[GP1:90,1] + 18.563;
   1:  PR[GP1:91,2] = PR[GP1:90,2] + -19.751;
   1:L PR[91] 10mm/sec CNT100;
   1:  PR[GP1:91,1] = PR[GP1:90,1] + 20.140;
   1:  PR[GP1:91,2] = PR[GP1:90,2] + -18.692;
   1:L PR[91] 10mm/sec CNT100;
